LIN {X 0,Y 210.674,Z 740.227,A -85,B 0,C 180,E1 4144.705,E2 4144.705} C_VEL
LIN {X 0,Y 221.818,Z 721.614,A -85,B 0,C 180,E1 4143.81,E2 4143.81} C_VEL
LIN {X 0,Y 225.35,Z 714.922,A -85,B 0,C 180,E1 4143.336,E2 4143.336} C_VEL
LIN {X 0,Y 232.907,Z 698.102,A -85,B 0,C 180,E1 4141.321,E2 4141.321} C_VEL
LIN {X 0,Y 235.66,Z 691.099,A -85,B 0,C 180,E1 4140.884,E2 4140.884} C_VEL
LIN {X 0,Y 242.843,Z 670.512,A -85,B 0,C 180,E1 4140.52,E2 4140.52} C_VEL
LIN {X 0,Y 247.959,Z 650.095,A -85,B 0,C 180,E1 4140.233,E2 4140.233} C_VEL
LIN {X 0,Y 251.406,Z 630.033,A -85,B 0,C 180,E1 4139.968,E2 4139.968} C_VEL
LIN {X 0,Y 253.666,Z 611.872,A -85,B 0,C 180,E1 4139.728,E2 4139.728} C_VEL
LIN {X 0,Y 254.145,Z 615.413,A -85,B 0,C 180,E1 4134.932,E2 4134.932} C_VEL
LIN {X 0,Y 255.029,Z 619.345,A -85,B 0,C 180,E1 4132.123,E2 4132.123} C_VEL
LIN {X 0,Y 260.484,Z 634.906,A -85,B 0,C 180,E1 4123.968,E2 4123.968} C_VEL
LIN {X 0,Y 268.032,Z 645.56,A -85,B 0,C 180,E1 4117.878,E2 4117.878} C_VEL
LIN {X 0,Y 279.58,Z 655.999,A -85,B 0,C 180,E1 4111.494,E2 4111.494} C_VEL
LIN {X 0,Y 288.035,Z 662.589,A -85,B 0,C 180,E1 4107.697,E2 4107.697} C_VEL
LIN {X 0,Y 293.255,Z 666.559,A -85,B 0,C 180,E1 4105.252,E2 4105.252} C_VEL
LIN {X 0,Y 299.992,Z 671.93,A -85,B 0,C 180,E1 4101.864,E2 4101.864} C_VEL
LIN {X 0,Y 304.317,Z 675.457,A -85,B 0,C 180,E1 4099.555,E2 4099.555} C_VEL
LIN {X 0,Y 310.73,Z 680.537,A -85,B 0,C 180,E1 4095.985,E2 4095.985} C_VEL
LIN {X 0,Y 314.599,Z 683.638,A -85,B 0,C 180,E1 4093.71,E2 4093.71} C_VEL
LIN {X 0,Y 320.356,Z 688.374,A -85,B 0,C 180,E1 4090.14,E2 4090.14} C_VEL
LIN {X 0,Y 324.684,Z 691.53,A -85,B 0,C 180,E1 4087.347,E2 4087.347} C_VEL
LIN {X 0,Y 329.45,Z 695.655,A -85,B 0,C 180,E1 4083.946,E2 4083.946} C_VEL
LIN {X 0,Y 334.291,Z 698.905,A -85,B 0,C 180,E1 4080.362,E2 4080.362} C_VEL
LIN {X 0,Y 336.58,Z 700.785,A -85,B 0,C 180,E1 4078.464,E2 4078.464} C_VEL
LIN {X 0,Y 340.334,Z 704.161,A -85,B 0,C 180,E1 4075.027,E2 4075.027} C_VEL
LIN {X 0,Y 343.918,Z 706.626,A -85,B 0,C 180,E1 4071.488,E2 4071.488} C_VEL
LIN {X 0,Y 347.168,Z 708.204,A -85,B 0,C 180,E1 4067.948,E2 4067.948} C_VEL
LIN {X 0,Y 348.332,Z 709.173,A -85,B 0,C 180,E1 4066.337,E2 4066.337} C_VEL
LIN {X 0,Y 350.261,Z 711.431,A -85,B 0,C 180,E1 4063.033,E2 4063.033} C_VEL
LIN {X 0,Y 351.887,Z 712.957,A -85,B 0,C 180,E1 4059.651,E2 4059.651} C_VEL
LIN {X 0,Y 353.094,Z 713.879,A -85,B 0,C 180,E1 4056.34,E2 4056.34} C_VEL
LIN {X 0,Y 353.771,Z 714.356,A -85,B 0,C 180,E1 4053.078,E2 4053.078} C_VEL
LIN {X 0,Y 353.955,Z 714.518,A -85,B 0,C 180,E1 4049.676,E2 4049.676} C_VEL
LIN {X 0,Y 353.709,Z 714.308,A -85,B 0,C 180,E1 4046.435,E2 4046.435} C_VEL
LIN {X 0,Y 352.933,Z 713.762,A -85,B 0,C 180,E1 4043.167,E2 4043.167} C_VEL
LIN {X 0,Y 351.648,Z 712.791,A -85,B 0,C 180,E1 4039.847,E2 4039.847} C_VEL
LIN {X 0,Y 349.965,Z 711.152,A -85,B 0,C 180,E1 4036.451,E2 4036.451} C_VEL
LIN {X 0,Y 347.988,Z 708.725,A -85,B 0,C 180,E1 4033.131,E2 4033.131} C_VEL
LIN {X 0,Y 345.166,Z 707.3,A -85,B 0,C 180,E1 4029.836,E2 4029.836} C_VEL
LIN {X 0,Y 341.961,Z 705.369,A -85,B 0,C 180,E1 4026.569,E2 4026.569} C_VEL
LIN {X 0,Y 338.532,Z 702.666,A -85,B 0,C 180,E1 4023.326,E2 4023.326} C_VEL
LIN {X 0,Y 334.734,Z 699.159,A -85,B 0,C 180,E1 4020.002,E2 4020.002} C_VEL
LIN {X 0,Y 330.098,Z 696.163,A -85,B 0,C 180,E1 4016.547,E2 4016.547} C_VEL
LIN {X 0,Y 325.217,Z 692.068,A -85,B 0,C 180,E1 4013.05,E2 4013.05} C_VEL
LIN {X 0,Y 322.331,Z 689.725,A -85,B 0,C 180,E1 4011.114,E2 4011.114} C_VEL
LIN {X 0,Y 316.916,Z 685.673,A -85,B 0,C 180,E1 4007.715,E2 4007.715} C_VEL
LIN {X 0,Y 311.447,Z 681.018,A -85,B 0,C 180,E1 4004.401,E2 4004.401} C_VEL
LIN {X 0,Y 305.202,Z 676.225,A -85,B 0,C 180,E1 4000.921,E2 4000.921} C_VEL
LIN {X 0,Y 300.242,Z 672.107,A -85,B 0,C 180,E1 3998.259,E2 3998.259} C_VEL
LIN {X 0,Y 293.548,Z 666.815,A -85,B 0,C 180,E1 3994.892,E2 3994.892} C_VEL
LIN {X 0,Y 288.653,Z 663.022,A -85,B 0,C 180,E1 3992.578,E2 3992.578} C_VEL
LIN {X 0,Y 280.59,Z 656.799,A -85,B 0,C 180,E1 3988.975,E2 3988.975} C_VEL
LIN {X 0,Y 270.966,Z 648.453,A -85,B 0,C 180,E1 3983.936,E2 3983.936} C_VEL
LIN {X 0,Y 263.336,Z 639.521,A -85,B 0,C 180,E1 3978.587,E2 3978.587} C_VEL
LIN {X 0,Y 257.411,Z 627.943,A -85,B 0,C 180,E1 3972.325,E2 3972.325} C_VEL
LIN {X 0,Y 254.738,Z 618.098,A -85,B 0,C 180,E1 3967.092,E2 3967.092} C_VEL
LIN {X 0,Y 253.972,Z 614.598,A -85,B 0,C 180,E1 3964.28,E2 3964.28} C_VEL
LIN {X 0,Y 253.666,Z 611.872,A -85,B 0,C 180,E1 3960.272,E2 3960.272} C_VEL
LIN {X 0,Y 249.3,Z 643.642,A -85,B 0,C 180,E1 3959.853,E2 3959.853} C_VEL
LIN {X 0,Y 244.621,Z 664.019,A -85,B 0,C 180,E1 3959.573,E2 3959.573} C_VEL
LIN {X 0,Y 238.978,Z 682.281,A -85,B 0,C 180,E1 3959.285,E2 3959.285} C_VEL
LIN {X 0,Y 230.509,Z 703.314,A -85,B 0,C 180,E1 3958.824,E2 3958.824} C_VEL
LIN {X 0,Y 222.058,Z 720.216,A -85,B 0,C 180,E1 3958.313,E2 3958.313} C_VEL
LIN {X 0,Y 211.154,Z 738.544,A -85,B 0,C 180,E1 3957.565,E2 3957.565} C_VEL
LIN {X 0,Y 199.308,Z 755.025,A -85,B 0,C 180,E1 3956.64,E2 3956.64} C_VEL
LIN {X 0,Y 188.015,Z 768.679,A -85,B 0,C 180,E1 3955.629,E2 3955.629} C_VEL
LIN {X 0,Y 173.879,Z 783.577,A -85,B 0,C 180,E1 3954.14,E2 3954.14} C_VEL
LIN {X 0,Y 159.406,Z 796.517,A -85,B 0,C 180,E1 3952.311,E2 3952.311} C_VEL
LIN {X 0,Y 146.082,Z 807.005,A -85,B 0,C 180,E1 3950.256,E2 3950.256} C_VEL
LIN {X 0,Y 129.637,Z 818.368,A -85,B 0,C 180,E1 3947.057,E2 3947.057} C_VEL
LIN {X 0,Y 113.071,Z 827.981,A -85,B 0,C 180,E1 3942.744,E2 3942.744} C_VEL
LIN {X 0,Y 99.321,Z 834.97,A -85,B 0,C 180,E1 3937.839,E2 3937.839} C_VEL
LIN {X 0,Y 83.5,Z 842.05,A -85,B 0,C 180,E1 3929.556,E2 3929.556} C_VEL
LIN {X 0,Y 69.946,Z 847.19,A -85,B 0,C 180,E1 3917.745,E2 3917.745} C_VEL
LIN {X 0,Y 61.606,Z 850.22,A -85,B 0,C 180,E1 3904.613,E2 3904.613} C_VEL
LIN {X 0,Y 56.485,Z 852.404,A -85,B 0,C 180,E1 3885.397,E2 3885.397} C_VEL
LIN {X 0,Y 56.061,Z 852.878,A -85,B 0,C 180,E1 3871.022,E2 3871.022} C_VEL
LIN {X 0,Y 56.17,Z 852.551,A -85,B 0,C 180,E1 3858.448,E2 3858.448} C_VEL
LIN {X 0,Y 60.475,Z 850.675,A -85,B 0,C 180,E1 3838.058,E2 3838.058} C_VEL
LIN {X 0,Y 68.915,Z 847.568,A -85,B 0,C 180,E1 3823.497,E2 3823.497} C_VEL
LIN {X 0,Y 79.87,Z 843.421,A -85,B 0,C 180,E1 3812.995,E2 3812.995} C_VEL
LIN {X 0,Y 95.202,Z 836.983,A -85,B 0,C 180,E1 3803.979,E2 3803.979} C_VEL
LIN {X 0,Y 111.312,Z 828.923,A -85,B 0,C 180,E1 3797.803,E2 3797.803} C_VEL
LIN {X 0,Y 125.885,Z 820.608,A -85,B 0,C 180,E1 3793.804,E2 3793.804} C_VEL
LIN {X 0,Y 143.255,Z 809.115,A -85,B 0,C 180,E1 3790.235,E2 3790.235} C_VEL
LIN {X 0,Y 157.491,Z 798.103,A -85,B 0,C 180,E1 3787.96,E2 3787.96} C_VEL
LIN {X 0,Y 170.969,Z 786.254,A -85,B 0,C 180,E1 3786.195,E2 3786.195} C_VEL
LIN {X 0,Y 186.547,Z 770.362,A -85,B 0,C 180,E1 3784.515,E2 3784.515} C_VEL
LIN {X 0,Y 198.324,Z 756.287,A -85,B 0,C 180,E1 3783.443,E2 3783.443} C_VEL
LIN {X 0,Y 209.671,Z 740.706,A -85,B 0,C 180,E1 3782.543,E2 3782.543} C_VEL
LIN {X 0,Y 221.065,Z 722.057,A -85,B 0,C 180,E1 3781.751,E2 3781.751} C_VEL
LIN {X 0,Y 229.514,Z 705.439,A -85,B 0,C 180,E1 3781.232,E2 3781.232} C_VEL
LIN {X 0,Y 235.66,Z 691.099,A -85,B 0,C 180,E1 3780.884,E2 3780.884} C_VEL
LIN {X 0,Y 238.036,Z 684.989,A -85,B 0,C 180,E1 3780.593,E2 3780.593} C_VEL
LIN {X 0,Y 244.118,Z 666.072,A -85,B 0,C 180,E1 3778.809,E2 3778.809} C_VEL
LIN {X 0,Y 246.08,Z 658.696,A -85,B 0,C 180,E1 3778.485,E2 3778.485} C_VEL
LIN {X 0,Y 250.367,Z 637.413,A -85,B 0,C 180,E1 3778.231,E2 3778.231} C_VEL
LIN {X 0,Y 252.664,Z 621.011,A -85,B 0,C 180,E1 3778.026,E2 3778.026} C_VEL
LIN {X 0,Y 253.065,Z 623.238,A -85,B 0,C 180,E1 3775.251,E2 3775.251} C_VEL
LIN {X 0,Y 253.864,Z 627.304,A -85,B 0,C 180,E1 3772.429,E2 3772.429} C_VEL
LIN {X 0,Y 258.424,Z 642.042,A -85,B 0,C 180,E1 3764.642,E2 3764.642} C_VEL
LIN {X 0,Y 265.618,Z 652.99,A -85,B 0,C 180,E1 3758.248,E2 3758.248} C_VEL
LIN {X 0,Y 276.691,Z 663.352,A -85,B 0,C 180,E1 3751.758,E2 3751.758} C_VEL
LIN {X 0,Y 286.024,Z 670.633,A -85,B 0,C 180,E1 3747.442,E2 3747.442} C_VEL
LIN {X 0,Y 291.129,Z 674.665,A -85,B 0,C 180,E1 3745.015,E2 3745.015} C_VEL
LIN {X 0,Y 297.886,Z 679.891,A -85,B 0,C 180,E1 3741.628,E2 3741.628} C_VEL
LIN {X 0,Y 304.458,Z 685.399,A -85,B 0,C 180,E1 3738.078,E2 3738.078} C_VEL
LIN {X 0,Y 310.736,Z 690.084,A -85,B 0,C 180,E1 3734.543,E2 3734.543} C_VEL
LIN {X 0,Y 316.536,Z 695.023,A -85,B 0,C 180,E1 3730.997,E2 3730.997} C_VEL
LIN {X 0,Y 321.866,Z 698.858,A -85,B 0,C 180,E1 3727.632,E2 3727.632} C_VEL
LIN {X 0,Y 326.947,Z 703.244,A -85,B 0,C 180,E1 3724.03,E2 3724.03} C_VEL
LIN {X 0,Y 331.613,Z 706.372,A -85,B 0,C 180,E1 3720.633,E2 3720.633} C_VEL
LIN {X 0,Y 333.853,Z 708.095,A -85,B 0,C 180,E1 3718.827,E2 3718.827} C_VEL
LIN {X 0,Y 337.827,Z 711.687,A -85,B 0,C 180,E1 3715.225,E2 3715.225} C_VEL
LIN {X 0,Y 341.357,Z 714.12,A -85,B 0,C 180,E1 3711.826,E2 3711.826} C_VEL
LIN {X 0,Y 344.675,Z 715.784,A -85,B 0,C 180,E1 3708.257,E2 3708.257} C_VEL
LIN {X 0,Y 345.95,Z 716.669,A -85,B 0,C 180,E1 3706.626,E2 3706.626} C_VEL
LIN {X 0,Y 347.815,Z 718.903,A -85,B 0,C 180,E1 3703.464,E2 3703.464} C_VEL
LIN {X 0,Y 349.513,Z 720.522,A -85,B 0,C 180,E1 3700.049,E2 3700.049} C_VEL
LIN {X 0,Y 350.807,Z 721.495,A -85,B 0,C 180,E1 3696.711,E2 3696.711} C_VEL
LIN {X 0,Y 351.51,Z 722.006,A -85,B 0,C 180,E1 3693.424,E2 3693.424} C_VEL
LIN {X 0,Y 351.766,Z 722.221,A -85,B 0,C 180,E1 3690,E2 3690} C_VEL
LIN {X 0,Y 351.591,Z 722.033,A -85,B 0,C 180,E1 3686.74,E2 3686.74} C_VEL
LIN {X 0,Y 350.787,Z 721.516,A -85,B 0,C 180,E1 3683.453,E2 3683.453} C_VEL
LIN {X 0,Y 349.505,Z 720.527,A -85,B 0,C 180,E1 3679.95,E2 3679.95} C_VEL
LIN {X 0,Y 347.971,Z 719.018,A -85,B 0,C 180,E1 3676.711,E2 3676.711} C_VEL
LIN {X 0,Y 345.922,Z 716.659,A -85,B 0,C 180,E1 3673.373,E2 3673.373} C_VEL
LIN {X 0,Y 344.622,Z 715.769,A -85,B 0,C 180,E1 3671.74,E2 3671.74} C_VEL
LIN {X 0,Y 341.289,Z 714.097,A -85,B 0,C 180,E1 3668.158,E2 3668.158} C_VEL
LIN {X 0,Y 337.789,Z 711.674,A -85,B 0,C 180,E1 3664.772,E2 3664.772} C_VEL
LIN {X 0,Y 334.098,Z 708.347,A -85,B 0,C 180,E1 3661.392,E2 3661.392} C_VEL
LIN {X 0,Y 331.89,Z 706.536,A -85,B 0,C 180,E1 3659.595,E2 3659.595} C_VEL
LIN {X 0,Y 327.39,Z 703.585,A -85,B 0,C 180,E1 3656.292,E2 3656.292} C_VEL
LIN {X 0,Y 322.48,Z 699.458,A -85,B 0,C 180,E1 3652.801,E2 3652.801} C_VEL
LIN {X 0,Y 319.198,Z 696.92,A -85,B 0,C 180,E1 3650.67,E2 3650.67} C_VEL
LIN {X 0,Y 313.547,Z 692.596,A -85,B 0,C 180,E1 3647.159,E2 3647.159} C_VEL
LIN {X 0,Y 308.746,Z 688.532,A -85,B 0,C 180,E1 3644.301,E2 3644.301} C_VEL
LIN {X 0,Y 302.375,Z 683.685,A -85,B 0,C 180,E1 3640.781,E2 3640.781} C_VEL
LIN {X 0,Y 297.355,Z 679.512,A -85,B 0,C 180,E1 3638.085,E2 3638.085} C_VEL
LIN {X 0,Y 290.395,Z 674.023,A -85,B 0,C 180,E1 3634.605,E2 3634.605} C_VEL
LIN {X 0,Y 284.812,Z 669.781,A -85,B 0,C 180,E1 3631.999,E2 3631.999} C_VEL
LIN {X 0,Y 272.035,Z 659.617,A -85,B 0,C 180,E1 3625.808,E2 3625.808} C_VEL
LIN {X 0,Y 261.158,Z 646.993,A -85,B 0,C 180,E1 3618.17,E2 3618.17} C_VEL
LIN {X 0,Y 255.873,Z 635.734,A -85,B 0,C 180,E1 3611.942,E2 3611.942} C_VEL
LIN {X 0,Y 253.53,Z 625.643,A -85,B 0,C 180,E1 3606.557,E2 3606.557} C_VEL
LIN {X 0,Y 252.891,Z 622.329,A -85,B 0,C 180,E1 3603.844,E2 3603.844} C_VEL
LIN {X 0,Y 252.634,Z 621.243,A -85,B 0,C 180,E1 3601.964,E2 3601.964} C_VEL
LIN {X 0,Y 248.718,Z 646.779,A -85,B 0,C 180,E1 3601.657,E2 3601.657} C_VEL
LIN {X 0,Y 244.033,Z 666.201,A -85,B 0,C 180,E1 3601.423,E2 3601.423} C_VEL
LIN {X 0,Y 237.507,Z 686.316,A -85,B 0,C 180,E1 3601.144,E2 3601.144} C_VEL
LIN {X 0,Y 229.482,Z 705.211,A -85,B 0,C 180,E1 3600.777,E2 3600.777} C_VEL
LIN {X 0,Y 220.465,Z 722.748,A -85,B 0,C 180,E1 3600.311,E2 3600.311} C_VEL
LIN {X 0,Y 208.618,Z 741.685,A -85,B 0,C 180,E1 3599.614,E2 3599.614} C_VEL
LIN {X 0,Y 197.505,Z 756.683,A -85,B 0,C 180,E1 3598.863,E2 3598.863} C_VEL
LIN {X 0,Y 184.072,Z 772.379,A -85,B 0,C 180,E1 3597.808,E2 3597.808} C_VEL
LIN {X 0,Y 169.299,Z 786.908,A -85,B 0,C 180,E1 3596.431,E2 3596.431} C_VEL
LIN {X 0,Y 155.594,Z 798.659,A -85,B 0,C 180,E1 3594.88,E2 3594.88} C_VEL
LIN {X 0,Y 138.984,Z 811.022,A -85,B 0,C 180,E1 3592.542,E2 3592.542} C_VEL
LIN {X 0,Y 122.989,Z 821.059,A -85,B 0,C 180,E1 3589.628,E2 3589.628} C_VEL
LIN {X 0,Y 108.169,Z 829.154,A -85,B 0,C 180,E1 3586.057,E2 3586.057} C_VEL
LIN {X 0,Y 90.447,Z 837.455,A -85,B 0,C 180,E1 3579.987,E2 3579.987} C_VEL
LIN {X 0,Y 74.938,Z 843.452,A -85,B 0,C 180,E1 3571.712,E2 3571.712} C_VEL
LIN {X 0,Y 62.908,Z 847.538,A -85,B 0,C 180,E1 3561.149,E2 3561.149} C_VEL
LIN {X 0,Y 52.118,Z 850.964,A -85,B 0,C 180,E1 3542.49,E2 3542.49} C_VEL
LIN {X 0,Y 48.181,Z 852.354,A -85,B 0,C 180,E1 3521.977,E2 3521.977} C_VEL
LIN {X 0,Y 48.051,Z 852.632,A -85,B 0,C 180,E1 3508.42,E2 3508.42} C_VEL
LIN {X 0,Y 49.054,Z 851.983,A -85,B 0,C 180,E1 3489.727,E2 3489.727} C_VEL
LIN {X 0,Y 55.075,Z 849.978,A -85,B 0,C 180,E1 3470.551,E2 3470.551} C_VEL
LIN {X 0,Y 64.861,Z 846.901,A -85,B 0,C 180,E1 3456.719,E2 3456.719} C_VEL
LIN {X 0,Y 79.842,Z 841.738,A -85,B 0,C 180,E1 3445.233,E2 3445.233} C_VEL
LIN {X 0,Y 96.521,Z 834.727,A -85,B 0,C 180,E1 3437.637,E2 3437.637} C_VEL
LIN {X 0,Y 110.912,Z 827.74,A -85,B 0,C 180,E1 3433.201,E2 3433.201} C_VEL
LIN {X 0,Y 127.705,Z 818.334,A -85,B 0,C 180,E1 3429.432,E2 3429.432} C_VEL
LIN {X 0,Y 144.922,Z 806.767,A -85,B 0,C 180,E1 3426.554,E2 3426.554} C_VEL
LIN {X 0,Y 159.497,Z 795.486,A -85,B 0,C 180,E1 3424.646,E2 3424.646} C_VEL
LIN {X 0,Y 176.194,Z 780.394,A -85,B 0,C 180,E1 3422.893,E2 3422.893} C_VEL
LIN {X 0,Y 189.058,Z 766.76,A -85,B 0,C 180,E1 3421.775,E2 3421.775} C_VEL
LIN {X 0,Y 201.986,Z 751.007,A -85,B 0,C 180,E1 3420.824,E2 3420.824} C_VEL
LIN {X 0,Y 213.963,Z 733.546,A -85,B 0,C 180,E1 3420.055,E2 3420.055} C_VEL
LIN {X 0,Y 222.968,Z 718.144,A -85,B 0,C 180,E1 3419.551,E2 3419.551} C_VEL
LIN {X 0,Y 231.988,Z 699.85,A -85,B 0,C 180,E1 3419.105,E2 3419.105} C_VEL
LIN {X 0,Y 239.765,Z 679.826,A -85,B 0,C 180,E1 3418.756,E2 3418.756} C_VEL
LIN {X 0,Y 245.667,Z 660.249,A -85,B 0,C 180,E1 3418.504,E2 3418.504} C_VEL
LIN {X 0,Y 246.08,Z 658.696,A -85,B 0,C 180,E1 3418.485,E2 3418.485} C_VEL
LIN {X 0,Y 247.29,Z 653.76,A -85,B 0,C 180,E1 3418.194,E2 3418.194} C_VEL
LIN {X 0,Y 250.073,Z 641.294,A -85,B 0,C 180,E1 3416.626,E2 3416.626} C_VEL
LIN {X 0,Y 250.775,Z 636.973,A -85,B 0,C 180,E1 3416.396,E2 3416.396} C_VEL
LIN {X 0,Y 251.823,Z 630.238,A -85,B 0,C 180,E1 3416.317,E2 3416.317} C_VEL
LIN {X 0,Y 252.307,Z 633.846,A -85,B 0,C 180,E1 3413.525,E2 3413.525} C_VEL
LIN {X 0,Y 256.15,Z 649.128,A -85,B 0,C 180,E1 3405.313,E2 3405.313} C_VEL
LIN {X 0,Y 263,Z 660.366,A -85,B 0,C 180,E1 3398.606,E2 3398.606} C_VEL
LIN {X 0,Y 282.175,Z 677.465,A -85,B 0,C 180,E1 3387.906,E2 3387.906} C_VEL
LIN {X 0,Y 287.738,Z 681.797,A -85,B 0,C 180,E1 3385.271,E2 3385.271} C_VEL
LIN {X 0,Y 294.58,Z 687.092,A -85,B 0,C 180,E1 3381.863,E2 3381.863} C_VEL
LIN {X 0,Y 301.39,Z 692.769,A -85,B 0,C 180,E1 3378.193,E2 3378.193} C_VEL
LIN {X 0,Y 308.027,Z 697.735,A -85,B 0,C 180,E1 3374.517,E2 3374.517} C_VEL
LIN {X 0,Y 314.137,Z 702.845,A -85,B 0,C 180,E1 3370.771,E2 3370.771} C_VEL
LIN {X 0,Y 319.077,Z 706.411,A -85,B 0,C 180,E1 3367.664,E2 3367.664} C_VEL
LIN {X 0,Y 323.715,Z 710.397,A -85,B 0,C 180,E1 3364.417,E2 3364.417} C_VEL
LIN {X 0,Y 328.566,Z 713.706,A -85,B 0,C 180,E1 3360.912,E2 3360.912} C_VEL
LIN {X 0,Y 330.854,Z 715.363,A -85,B 0,C 180,E1 3359.113,E2 3359.113} C_VEL
LIN {X 0,Y 334.802,Z 718.941,A -85,B 0,C 180,E1 3355.617,E2 3355.617} C_VEL
LIN {X 0,Y 338.558,Z 721.576,A -85,B 0,C 180,E1 3352.007,E2 3352.007} C_VEL
LIN {X 0,Y 341.818,Z 723.237,A -85,B 0,C 180,E1 3348.592,E2 3348.592} C_VEL
LIN {X 0,Y 343.348,Z 724.234,A -85,B 0,C 180,E1 3346.689,E2 3346.689} C_VEL
LIN {X 0,Y 345.306,Z 726.538,A -85,B 0,C 180,E1 3343.394,E2 3343.394} C_VEL
LIN {X 0,Y 346.929,Z 728.083,A -85,B 0,C 180,E1 3340.125,E2 3340.125} C_VEL
LIN {X 0,Y 348.245,Z 729.07,A -85,B 0,C 180,E1 3336.76,E2 3336.76} C_VEL
LIN {X 0,Y 348.97,Z 729.591,A -85,B 0,C 180,E1 3333.449,E2 3333.449} C_VEL
LIN {X 0,Y 349.227,Z 729.808,A -85,B 0,C 180,E1 3330,E2 3330} C_VEL
LIN {X 0,Y 349.044,Z 729.616,A -85,B 0,C 180,E1 3326.716,E2 3326.716} C_VEL
LIN {X 0,Y 348.22,Z 729.081,A -85,B 0,C 180,E1 3323.357,E2 3323.357} C_VEL
LIN {X 0,Y 347.033,Z 728.155,A -85,B 0,C 180,E1 3320.046,E2 3320.046} C_VEL
LIN {X 0,Y 345.409,Z 726.629,A -85,B 0,C 180,E1 3316.781,E2 3316.781} C_VEL
LIN {X 0,Y 343.365,Z 724.308,A -85,B 0,C 180,E1 3313.42,E2 3313.42} C_VEL
LIN {X 0,Y 342.086,Z 723.358,A -85,B 0,C 180,E1 3311.754,E2 3311.754} C_VEL
LIN {X 0,Y 339.141,Z 721.922,A -85,B 0,C 180,E1 3308.558,E2 3308.558} C_VEL
LIN {X 0,Y 335.405,Z 719.421,A -85,B 0,C 180,E1 3304.957,E2 3304.957} C_VEL
LIN {X 0,Y 331.598,Z 716.116,A -85,B 0,C 180,E1 3301.55,E2 3301.55} C_VEL
LIN {X 0,Y 329.152,Z 714.04,A -85,B 0,C 180,E1 3299.517,E2 3299.517} C_VEL
LIN {X 0,Y 324.617,Z 711.095,A -85,B 0,C 180,E1 3296.247,E2 3296.247} C_VEL
LIN {X 0,Y 319.801,Z 707.113,A -85,B 0,C 180,E1 3292.851,E2 3292.851} C_VEL
LIN {X 0,Y 316.533,Z 704.497,A -85,B 0,C 180,E1 3290.688,E2 3290.688} C_VEL
LIN {X 0,Y 310.786,Z 700.181,A -85,B 0,C 180,E1 3287.166,E2 3287.166} C_VEL
LIN {X 0,Y 305.337,Z 695.643,A -85,B 0,C 180,E1 3283.949,E2 3283.949} C_VEL
LIN {X 0,Y 298.936,Z 690.73,A -85,B 0,C 180,E1 3280.442,E2 3280.442} C_VEL
LIN {X 0,Y 294.204,Z 686.831,A -85,B 0,C 180,E1 3277.948,E2 3277.948} C_VEL
LIN {X 0,Y 287.367,Z 681.475,A -85,B 0,C 180,E1 3274.537,E2 3274.537} C_VEL
LIN {X 0,Y 282.161,Z 677.461,A -85,B 0,C 180,E1 3272.096,E2 3272.096} C_VEL
LIN {X 0,Y 269.586,Z 667.398,A -85,B 0,C 180,E1 3265.823,E2 3265.823} C_VEL
LIN {X 0,Y 258.829,Z 654.428,A -85,B 0,C 180,E1 3257.757,E2 3257.757} C_VEL
LIN {X 0,Y 253.962,Z 642.615,A -85,B 0,C 180,E1 3251.112,E2 3251.112} C_VEL
LIN {X 0,Y 252.196,Z 633.003,A -85,B 0,C 180,E1 3245.906,E2 3245.906} C_VEL
LIN {X 0,Y 251.811,Z 630.349,A -85,B 0,C 180,E1 3243.676,E2 3243.676} C_VEL
LIN {X 0,Y 248.294,Z 650.213,A -85,B 0,C 180,E1 3243.465,E2 3243.465} C_VEL
LIN {X 0,Y 242.944,Z 670.96,A -85,B 0,C 180,E1 3243.255,E2 3243.255} C_VEL
LIN {X 0,Y 235.786,Z 691.065,A -85,B 0,C 180,E1 3243.015,E2 3243.015} C_VEL
LIN {X 0,Y 228.219,Z 708.169,A -85,B 0,C 180,E1 3242.725,E2 3242.725} C_VEL
LIN {X 0,Y 217.495,Z 727.891,A -85,B 0,C 180,E1 3242.265,E2 3242.265} C_VEL
LIN {X 0,Y 207.061,Z 743.799,A -85,B 0,C 180,E1 3241.749,E2 3241.749} C_VEL
LIN {X 0,Y 195,Z 759.6,A -85,B 0,C 180,E1 3241.062,E2 3241.062} C_VEL
LIN {X 0,Y 180.469,Z 775.658,A -85,B 0,C 180,E1 3240.092,E2 3240.092} C_VEL
LIN {X 0,Y 166.996,Z 788.453,A -85,B 0,C 180,E1 3239.019,E2 3239.019} C_VEL
LIN {X 0,Y 151.122,Z 801.569,A -85,B 0,C 180,E1 3237.466,E2 3237.466} C_VEL
LIN {X 0,Y 134.41,Z 813.162,A -85,B 0,C 180,E1 3235.402,E2 3235.402} C_VEL
LIN {X 0,Y 118.889,Z 822.451,A -85,B 0,C 180,E1 3232.911,E2 3232.911} C_VEL
LIN {X 0,Y 100.851,Z 831.67,A -85,B 0,C 180,E1 3228.956,E2 3228.956} C_VEL
LIN {X 0,Y 83.492,Z 838.899,A -85,B 0,C 180,E1 3223.337,E2 3223.337} C_VEL
LIN {X 0,Y 68.829,Z 844.066,A -85,B 0,C 180,E1 3215.962,E2 3215.962} C_VEL
LIN {X 0,Y 52.656,Z 848.823,A -85,B 0,C 180,E1 3201.123,E2 3201.123} C_VEL
LIN {X 0,Y 43.384,Z 851.188,A -85,B 0,C 180,E1 3182.009,E2 3182.009} C_VEL
LIN {X 0,Y 40.091,Z 852.214,A -85,B 0,C 180,E1 3160.054,E2 3160.054} C_VEL
LIN {X 0,Y 40.029,Z 852.374,A -85,B 0,C 180,E1 3147.137,E2 3147.137} C_VEL
LIN {X 0,Y 42.07,Z 851.558,A -85,B 0,C 180,E1 3123.157,E2 3123.157} C_VEL
LIN {X 0,Y 49.881,Z 849.513,A -85,B 0,C 180,E1 3103.027,E2 3103.027} C_VEL
LIN {X 0,Y 62.065,Z 846.165,A -85,B 0,C 180,E1 3088.944,E2 3088.944} C_VEL
LIN {X 0,Y 79.965,Z 840.246,A -85,B 0,C 180,E1 3078.148,E2 3078.148} C_VEL
LIN {X 0,Y 95.278,Z 834.085,A -85,B 0,C 180,E1 3072.598,E2 3072.598} C_VEL
LIN {X 0,Y 111.231,Z 826.559,A -85,B 0,C 180,E1 3068.598,E2 3068.598} C_VEL
LIN {X 0,Y 130.508,Z 815.646,A -85,B 0,C 180,E1 3065.166,E2 3065.166} C_VEL
LIN {X 0,Y 145.517,Z 805.602,A -85,B 0,C 180,E1 3063.168,E2 3063.168} C_VEL
LIN {X 0,Y 162.034,Z 792.845,A -85,B 0,C 180,E1 3061.43,E2 3061.43} C_VEL
LIN {X 0,Y 177.559,Z 778.57,A -85,B 0,C 180,E1 3060.123,E2 3060.123} C_VEL
LIN {X 0,Y 190.53,Z 764.791,A -85,B 0,C 180,E1 3059.214,E2 3059.214} C_VEL
LIN {X 0,Y 204.546,Z 747.356,A -85,B 0,C 180,E1 3058.387,E2 3058.387} C_VEL
LIN {X 0,Y 215.619,Z 730.893,A -85,B 0,C 180,E1 3057.82,E2 3057.82} C_VEL
LIN {X 0,Y 225.698,Z 713.295,A -85,B 0,C 180,E1 3057.378,E2 3057.378} C_VEL
LIN {X 0,Y 234.777,Z 693.553,A -85,B 0,C 180,E1 3057.021,E2 3057.021} C_VEL
LIN {X 0,Y 241.336,Z 675.883,A -85,B 0,C 180,E1 3056.796,E2 3056.796} C_VEL
LIN {X 0,Y 247.442,Z 654.174,A -85,B 0,C 180,E1 3056.576,E2 3056.576} C_VEL
LIN {X 0,Y 250.775,Z 636.973,A -85,B 0,C 180,E1 3056.396,E2 3056.396} C_VEL
LIN {X 0,Y 251.008,Z 635.871,A -85,B 0,C 180,E1 3056.158,E2 3056.158} C_VEL
LIN {X 0,Y 251.231,Z 635.803,A -85,B 0,C 180,E1 3055.473,E2 3055.473} C_VEL
LIN {X 0,Y 251.312,Z 637.609,A -85,B 0,C 180,E1 3054.477,E2 3054.477} C_VEL
LIN {X 0,Y 251.28,Z 645.589,A -85,B 0,C 180,E1 3051.782,E2 3051.782} C_VEL
LIN {X 0,Y 251.36,Z 646.438,A -85,B 0,C 180,E1 3051.363,E2 3051.363} C_VEL
LIN {X 0,Y 254.203,Z 657.281,A -85,B 0,C 180,E1 3045.315,E2 3045.315} C_VEL
LIN {X 0,Y 260.03,Z 667.519,A -85,B 0,C 180,E1 3039.059,E2 3039.059} C_VEL
LIN {X 0,Y 270.301,Z 677.852,A -85,B 0,C 180,E1 3032.232,E2 3032.232} C_VEL
LIN {X 0,Y 282.152,Z 687.144,A -85,B 0,C 180,E1 3026.453,E2 3026.453} C_VEL
LIN {X 0,Y 289.105,Z 692.824,A -85,B 0,C 180,E1 3023.017,E2 3023.017} C_VEL
LIN {X 0,Y 294.362,Z 696.919,A -85,B 0,C 180,E1 3020.329,E2 3020.329} C_VEL
LIN {X 0,Y 301.066,Z 702.252,A -85,B 0,C 180,E1 3016.66,E2 3016.66} C_VEL
LIN {X 0,Y 305.071,Z 705.329,A -85,B 0,C 180,E1 3014.415,E2 3014.415} C_VEL
LIN {X 0,Y 310.84,Z 710.095,A -85,B 0,C 180,E1 3010.912,E2 3010.912} C_VEL
LIN {X 0,Y 315.67,Z 713.531,A -85,B 0,C 180,E1 3007.913,E2 3007.913} C_VEL
LIN {X 0,Y 320.47,Z 717.665,A -85,B 0,C 180,E1 3004.566,E2 3004.566} C_VEL
LIN {X 0,Y 325.452,Z 721.055,A -85,B 0,C 180,E1 3001.024,E2 3001.024} C_VEL
LIN {X 0,Y 327.786,Z 722.736,A -85,B 0,C 180,E1 2999.212,E2 2999.212} C_VEL
LIN {X 0,Y 331.716,Z 726.305,A -85,B 0,C 180,E1 2995.704,E2 2995.704} C_VEL
LIN {X 0,Y 335.545,Z 728.983,A -85,B 0,C 180,E1 2992.052,E2 2992.052} C_VEL
LIN {X 0,Y 338.929,Z 730.698,A -85,B 0,C 180,E1 2988.578,E2 2988.578} C_VEL
LIN {X 0,Y 340.381,Z 731.645,A -85,B 0,C 180,E1 2986.781,E2 2986.781} C_VEL
LIN {X 0,Y 342.471,Z 734.047,A -85,B 0,C 180,E1 2983.335,E2 2983.335} C_VEL
LIN {X 0,Y 344.087,Z 735.588,A -85,B 0,C 180,E1 2979.977,E2 2979.977} C_VEL
LIN {X 0,Y 345.408,Z 736.585,A -85,B 0,C 180,E1 2976.482,E2 2976.482} C_VEL
LIN {X 0,Y 346.13,Z 737.076,A -85,B 0,C 180,E1 2973.312,E2 2973.312} C_VEL
LIN {X 0,Y 346.351,Z 737.273,A -85,B 0,C 180,E1 2970,E2 2970} C_VEL
LIN {X 0,Y 346.165,Z 737.091,A -85,B 0,C 180,E1 2966.854,E2 2966.854} C_VEL
LIN {X 0,Y 345.392,Z 736.588,A -85,B 0,C 180,E1 2963.518,E2 2963.518} C_VEL
LIN {X 0,Y 344.271,Z 735.7,A -85,B 0,C 180,E1 2960.303,E2 2960.303} C_VEL
LIN {X 0,Y 342.6,Z 734.203,A -85,B 0,C 180,E1 2957.014,E2 2957.014} C_VEL
LIN {X 0,Y 340.639,Z 731.993,A -85,B 0,C 180,E1 2953.634,E2 2953.634} C_VEL
LIN {X 0,Y 339.482,Z 730.93,A -85,B 0,C 180,E1 2951.986,E2 2951.986} C_VEL
LIN {X 0,Y 336.314,Z 729.439,A -85,B 0,C 180,E1 2948.734,E2 2948.734} C_VEL
LIN {X 0,Y 332.552,Z 726.969,A -85,B 0,C 180,E1 2945.108,E2 2945.108} C_VEL
LIN {X 0,Y 328.912,Z 723.869,A -85,B 0,C 180,E1 2941.809,E2 2941.809} C_VEL
LIN {X 0,Y 326.09,Z 721.427,A -85,B 0,C 180,E1 2939.475,E2 2939.475} C_VEL
LIN {X 0,Y 321.434,Z 718.407,A -85,B 0,C 180,E1 2936.134,E2 2936.134} C_VEL
LIN {X 0,Y 316.466,Z 714.306,A -85,B 0,C 180,E1 2932.656,E2 2932.656} C_VEL
LIN {X 0,Y 313.291,Z 711.785,A -85,B 0,C 180,E1 2930.574,E2 2930.574} C_VEL
LIN {X 0,Y 307.417,Z 707.395,A -85,B 0,C 180,E1 2927.021,E2 2927.021} C_VEL
LIN {X 0,Y 302.285,Z 703.076,A -85,B 0,C 180,E1 2923.981,E2 2923.981} C_VEL
LIN {X 0,Y 295.781,Z 698.16,A -85,B 0,C 180,E1 2920.454,E2 2920.454} C_VEL
LIN {X 0,Y 290.499,Z 693.827,A -85,B 0,C 180,E1 2917.664,E2 2917.664} C_VEL
LIN {X 0,Y 283.328,Z 688.17,A -85,B 0,C 180,E1 2914.119,E2 2914.119} C_VEL
LIN {X 0,Y 278.041,Z 684.177,A -85,B 0,C 180,E1 2911.657,E2 2911.657} C_VEL
LIN {X 0,Y 262.385,Z 670.162,A -85,B 0,C 180,E1 2902.742,E2 2902.742} C_VEL
LIN {X 0,Y 256.199,Z 661.62,A -85,B 0,C 180,E1 2897.242,E2 2897.242} C_VEL
LIN {X 0,Y 251.997,Z 650.11,A -85,B 0,C 180,E1 2890.621,E2 2890.621} C_VEL
LIN {X 0,Y 250.829,Z 640.57,A -85,B 0,C 180,E1 2885.401,E2 2885.401} C_VEL
LIN {X 0,Y 245.941,Z 662.213,A -85,B 0,C 180,E1 2885.207,E2 2885.207} C_VEL
LIN {X 0,Y 239.89,Z 681.604,A -85,B 0,C 180,E1 2885.049,E2 2885.049} C_VEL
LIN {X 0,Y 231.276,Z 702.629,A -85,B 0,C 180,E1 2884.814,E2 2884.814} C_VEL
LIN {X 0,Y 222.299,Z 720.186,A -85,B 0,C 180,E1 2884.535,E2 2884.535} C_VEL
LIN {X 0,Y 210.503,Z 739.297,A -85,B 0,C 180,E1 2884.103,E2 2884.103} C_VEL
LIN {X 0,Y 198.354,Z 755.584,A -85,B 0,C 180,E1 2883.585,E2 2883.585} C_VEL
LIN {X 0,Y 184.704,Z 771.333,A -85,B 0,C 180,E1 2882.897,E2 2882.897} C_VEL
LIN {X 0,Y 169.069,Z 786.433,A -85,B 0,C 180,E1 2881.949,E2 2881.949} C_VEL
LIN {X 0,Y 154.993,Z 798.185,A -85,B 0,C 180,E1 2880.905,E2 2880.905} C_VEL
LIN {X 0,Y 136.989,Z 811.06,A -85,B 0,C 180,E1 2879.218,E2 2879.218} C_VEL
LIN {X 0,Y 119.872,Z 821.265,A -85,B 0,C 180,E1 2877.111,E2 2877.111} C_VEL
LIN {X 0,Y 102.509,Z 830.09,A -85,B 0,C 180,E1 2874.193,E2 2874.193} C_VEL
LIN {X 0,Y 83.39,Z 837.984,A -85,B 0,C 180,E1 2869.472,E2 2869.472} C_VEL
LIN {X 0,Y 67.799,Z 843.242,A -85,B 0,C 180,E1 2863.447,E2 2863.447} C_VEL
LIN {X 0,Y 51.757,Z 847.692,A -85,B 0,C 180,E1 2852.7,E2 2852.7} C_VEL
LIN {X 0,Y 37.717,Z 850.761,A -85,B 0,C 180,E1 2831.507,E2 2831.507} C_VEL
LIN {X 0,Y 32.267,Z 851.943,A -85,B 0,C 180,E1 2804.353,E2 2804.353} C_VEL
LIN {X 0,Y 32.046,Z 852.168,A -85,B 0,C 180,E1 2788.212,E2 2788.212} C_VEL
LIN {X 0,Y 34.631,Z 851.411,A -85,B 0,C 180,E1 2758.689,E2 2758.689} C_VEL
LIN {X 0,Y 44.375,Z 849.344,A -85,B 0,C 180,E1 2735.793,E2 2735.793} C_VEL
LIN {X 0,Y 58.264,Z 845.994,A -85,B 0,C 180,E1 2722.08,E2 2722.08} C_VEL
LIN {X 0,Y 77.797,Z 840.006,A -85,B 0,C 180,E1 2712.385,E2 2712.385} C_VEL
LIN {X 0,Y 93.829,Z 833.846,A -85,B 0,C 180,E1 2707.694,E2 2707.694} C_VEL
LIN {X 0,Y 111.282,Z 825.849,A -85,B 0,C 180,E1 2704.214,E2 2704.214} C_VEL
LIN {X 0,Y 130.026,Z 815.407,A -85,B 0,C 180,E1 2701.568,E2 2701.568} C_VEL
LIN {X 0,Y 145.975,Z 804.886,A -85,B 0,C 180,E1 2699.882,E2 2699.882} C_VEL
LIN {X 0,Y 163.03,Z 791.771,A -85,B 0,C 180,E1 2698.473,E2 2698.473} C_VEL
LIN {X 0,Y 178.142,Z 777.924,A -85,B 0,C 180,E1 2697.475,E2 2697.475} C_VEL
LIN {X 0,Y 191.274,Z 764.045,A -85,B 0,C 180,E1 2696.755,E2 2696.755} C_VEL
LIN {X 0,Y 205.44,Z 746.412,A -85,B 0,C 180,E1 2696.103,E2 2696.103} C_VEL
LIN {X 0,Y 216.077,Z 730.659,A -85,B 0,C 180,E1 2695.681,E2 2695.681} C_VEL
LIN {X 0,Y 226.209,Z 713.053,A -85,B 0,C 180,E1 2695.339,E2 2695.339} C_VEL
LIN {X 0,Y 235.332,Z 693.321,A -85,B 0,C 180,E1 2695.066,E2 2695.066} C_VEL
LIN {X 0,Y 241.917,Z 675.658,A -85,B 0,C 180,E1 2694.897,E2 2694.897} C_VEL
LIN {X 0,Y 248.045,Z 653.984,A -85,B 0,C 180,E1 2694.726,E2 2694.726} C_VEL
LIN {X 0,Y 250.827,Z 640.601,A -85,B 0,C 180,E1 2694.578,E2 2694.578} C_VEL
LIN {X 0,Y 251.36,Z 646.438,A -85,B 0,C 180,E1 2691.363,E2 2691.363} C_VEL
LIN {X 0,Y 251.633,Z 650.208,A -85,B 0,C 180,E1 2689.822,E2 2689.822} C_VEL
LIN {X 0,Y 251.84,Z 663.238,A -85,B 0,C 180,E1 2686.023,E2 2686.023} C_VEL
LIN {X 0,Y 252.409,Z 666.32,A -85,B 0,C 180,E1 2684.694,E2 2684.694} C_VEL
LIN {X 0,Y 257.161,Z 674.934,A -85,B 0,C 180,E1 2679.291,E2 2679.291} C_VEL
LIN {X 0,Y 274.549,Z 691.382,A -85,B 0,C 180,E1 2668.384,E2 2668.384} C_VEL
LIN {X 0,Y 279.83,Z 695.427,A -85,B 0,C 180,E1 2665.89,E2 2665.89} C_VEL
LIN {X 0,Y 286.84,Z 700.928,A -85,B 0,C 180,E1 2662.424,E2 2662.424} C_VEL
LIN {X 0,Y 291.315,Z 704.57,A -85,B 0,C 180,E1 2660.087,E2 2660.087} C_VEL
LIN {X 0,Y 298.145,Z 709.837,A -85,B 0,C 180,E1 2656.415,E2 2656.415} C_VEL
LIN {X 0,Y 302.844,Z 713.661,A -85,B 0,C 180,E1 2653.71,E2 2653.71} C_VEL
LIN {X 0,Y 308.776,Z 718.29,A -85,B 0,C 180,E1 2650.118,E2 2650.118} C_VEL
LIN {X 0,Y 312.473,Z 721.005,A -85,B 0,C 180,E1 2647.8,E2 2647.8} C_VEL
LIN {X 0,Y 317.388,Z 725.148,A -85,B 0,C 180,E1 2644.394,E2 2644.394} C_VEL
LIN {X 0,Y 322.426,Z 728.504,A -85,B 0,C 180,E1 2640.819,E2 2640.819} C_VEL
LIN {X 0,Y 324.828,Z 730.417,A -85,B 0,C 180,E1 2638.898,E2 2638.898} C_VEL
LIN {X 0,Y 328.525,Z 733.693,A -85,B 0,C 180,E1 2635.605,E2 2635.605} C_VEL
LIN {X 0,Y 332.479,Z 736.403,A -85,B 0,C 180,E1 2631.894,E2 2631.894} C_VEL
LIN {X 0,Y 335.583,Z 737.964,A -85,B 0,C 180,E1 2628.689,E2 2628.689} C_VEL
LIN {X 0,Y 337.049,Z 738.884,A -85,B 0,C 180,E1 2626.9,E2 2626.9} C_VEL
LIN {X 0,Y 339.152,Z 741.31,A -85,B 0,C 180,E1 2623.424,E2 2623.424} C_VEL
LIN {X 0,Y 340.756,Z 742.842,A -85,B 0,C 180,E1 2620.14,E2 2620.14} C_VEL
LIN {X 0,Y 342.142,Z 743.882,A -85,B 0,C 180,E1 2616.544,E2 2616.544} C_VEL
LIN {X 0,Y 342.873,Z 744.38,A -85,B 0,C 180,E1 2613.511,E2 2613.511} C_VEL
LIN {X 0,Y 343.14,Z 744.6,A -85,B 0,C 180,E1 2610,E2 2610} C_VEL
LIN {X 0,Y 342.951,Z 744.432,A -85,B 0,C 180,E1 2606.992,E2 2606.992} C_VEL
LIN {X 0,Y 342.126,Z 743.883,A -85,B 0,C 180,E1 2603.437,E2 2603.437} C_VEL
LIN {X 0,Y 340.929,Z 742.952,A -85,B 0,C 180,E1 2600.132,E2 2600.132} C_VEL
LIN {X 0,Y 339.165,Z 741.353,A -85,B 0,C 180,E1 2596.707,E2 2596.707} C_VEL
LIN {X 0,Y 337.162,Z 739.033,A -85,B 0,C 180,E1 2593.268,E2 2593.268} C_VEL
LIN {X 0,Y 335.714,Z 738.026,A -85,B 0,C 180,E1 2591.418,E2 2591.418} C_VEL
LIN {X 0,Y 332.577,Z 736.47,A -85,B 0,C 180,E1 2588.245,E2 2588.245} C_VEL
LIN {X 0,Y 328.699,Z 733.842,A -85,B 0,C 180,E1 2584.587,E2 2584.587} C_VEL
LIN {X 0,Y 324.974,Z 730.573,A -85,B 0,C 180,E1 2581.243,E2 2581.243} C_VEL
LIN {X 0,Y 322.76,Z 728.697,A -85,B 0,C 180,E1 2579.429,E2 2579.429} C_VEL
LIN {X 0,Y 318.055,Z 725.651,A -85,B 0,C 180,E1 2576.071,E2 2576.071} C_VEL
LIN {X 0,Y 313.109,Z 721.612,A -85,B 0,C 180,E1 2572.648,E2 2572.648} C_VEL
LIN {X 0,Y 309.771,Z 718.948,A -85,B 0,C 180,E1 2570.465,E2 2570.465} C_VEL
LIN {X 0,Y 303.624,Z 714.339,A -85,B 0,C 180,E1 2566.769,E2 2566.769} C_VEL
LIN {X 0,Y 298.643,Z 710.173,A -85,B 0,C 180,E1 2563.855,E2 2563.855} C_VEL
LIN {X 0,Y 291.703,Z 704.893,A -85,B 0,C 180,E1 2560.106,E2 2560.106} C_VEL
LIN {X 0,Y 286.862,Z 700.938,A -85,B 0,C 180,E1 2557.573,E2 2557.573} C_VEL
LIN {X 0,Y 279.393,Z 695.04,A -85,B 0,C 180,E1 2553.878,E2 2553.878} C_VEL
LIN {X 0,Y 264.968,Z 683.474,A -85,B 0,C 180,E1 2546.428,E2 2546.428} C_VEL
LIN {X 0,Y 253.746,Z 669.499,A -85,B 0,C 180,E1 2537.178,E2 2537.178} C_VEL
LIN {X 0,Y 249.836,Z 657.241,A -85,B 0,C 180,E1 2529.957,E2 2529.957} C_VEL
LIN {X 0,Y 249.23,Z 652.292,A -85,B 0,C 180,E1 2527.124,E2 2527.124} C_VEL
LIN {X 0,Y 243.27,Z 673.946,A -85,B 0,C 180,E1 2526.997,E2 2526.997} C_VEL
LIN {X 0,Y 236.667,Z 691.844,A -85,B 0,C 180,E1 2526.886,E2 2526.886} C_VEL
LIN {X 0,Y 228.023,Z 710.832,A -85,B 0,C 180,E1 2526.709,E2 2526.709} C_VEL
LIN {X 0,Y 217.342,Z 729.619,A -85,B 0,C 180,E1 2526.459,E2 2526.459} C_VEL
LIN {X 0,Y 206.657,Z 745.469,A -85,B 0,C 180,E1 2526.157,E2 2526.157} C_VEL
LIN {X 0,Y 192.412,Z 763.25,A -85,B 0,C 180,E1 2525.682,E2 2525.682} C_VEL
LIN {X 0,Y 178.572,Z 777.801,A -85,B 0,C 180,E1 2525.125,E2 2525.125} C_VEL
LIN {X 0,Y 162.436,Z 792.371,A -85,B 0,C 180,E1 2524.33,E2 2524.33} C_VEL
LIN {X 0,Y 146.221,Z 804.649,A -85,B 0,C 180,E1 2523.323,E2 2523.323} C_VEL
LIN {X 0,Y 130.06,Z 815.167,A -85,B 0,C 180,E1 2522.043,E2 2522.043} C_VEL
LIN {X 0,Y 109.981,Z 826.082,A -85,B 0,C 180,E1 2519.89,E2 2519.89} C_VEL
LIN {X 0,Y 93.085,Z 833.607,A -85,B 0,C 180,E1 2517.326,E2 2517.326} C_VEL
LIN {X 0,Y 74.526,Z 840.438,A -85,B 0,C 180,E1 2513.105,E2 2513.105} C_VEL
LIN {X 0,Y 54.789,Z 845.967,A -85,B 0,C 180,E1 2505.279,E2 2505.279} C_VEL
LIN {X 0,Y 39.345,Z 849.258,A -85,B 0,C 180,E1 2492.801,E2 2492.801} C_VEL
LIN {X 0,Y 26.541,Z 851.459,A -85,B 0,C 180,E1 2463.864,E2 2463.864} C_VEL
LIN {X 0,Y 24.073,Z 851.952,A -85,B 0,C 180,E1 2430,E2 2430} C_VEL
LIN {X 0,Y 27.056,Z 851.358,A -85,B 0,C 180,E1 2393.754,E2 2393.754} C_VEL
LIN {X 0,Y 39.345,Z 849.258,A -85,B 0,C 180,E1 2367.199,E2 2367.199} C_VEL
LIN {X 0,Y 54.789,Z 845.967,A -85,B 0,C 180,E1 2354.721,E2 2354.721} C_VEL
LIN {X 0,Y 74.526,Z 840.438,A -85,B 0,C 180,E1 2346.895,E2 2346.895} C_VEL
LIN {X 0,Y 93.085,Z 833.607,A -85,B 0,C 180,E1 2342.674,E2 2342.674} C_VEL
LIN {X 0,Y 110.981,Z 825.611,A -85,B 0,C 180,E1 2339.984,E2 2339.984} C_VEL
LIN {X 0,Y 130.06,Z 815.167,A -85,B 0,C 180,E1 2337.957,E2 2337.957} C_VEL
LIN {X 0,Y 146.221,Z 804.649,A -85,B 0,C 180,E1 2336.677,E2 2336.677} C_VEL
LIN {X 0,Y 163.45,Z 791.531,A -85,B 0,C 180,E1 2335.615,E2 2335.615} C_VEL
LIN {X 0,Y 178.685,Z 777.689,A -85,B 0,C 180,E1 2334.87,E2 2334.87} C_VEL
LIN {X 0,Y 191.978,Z 763.728,A -85,B 0,C 180,E1 2334.334,E2 2334.334} C_VEL
LIN {X 0,Y 206.148,Z 746.18,A -85,B 0,C 180,E1 2333.859,E2 2333.859} C_VEL
LIN {X 0,Y 216.834,Z 730.425,A -85,B 0,C 180,E1 2333.553,E2 2333.553} C_VEL
LIN {X 0,Y 227.006,Z 712.81,A -85,B 0,C 180,E1 2333.312,E2 2333.312} C_VEL
LIN {X 0,Y 236.159,Z 693.089,A -85,B 0,C 180,E1 2333.123,E2 2333.123} C_VEL
LIN {X 0,Y 243.017,Z 674.689,A -85,B 0,C 180,E1 2333.006,E2 2333.006} C_VEL
LIN {X 0,Y 249.183,Z 652.509,A -85,B 0,C 180,E1 2332.877,E2 2332.877} C_VEL
LIN {X 0,Y 249.274,Z 652.11,A -85,B 0,C 180,E1 2332.868,E2 2332.868} C_VEL
LIN {X 0,Y 251.565,Z 664.276,A -85,B 0,C 180,E1 2325.98,E2 2325.98} C_VEL
LIN {X 0,Y 252.409,Z 666.32,A -85,B 0,C 180,E1 2324.694,E2 2324.694} C_VEL
LIN {X 0,Y 253.298,Z 670.474,A -85,B 0,C 180,E1 2322.931,E2 2322.931} C_VEL
LIN {X 0,Y 254.779,Z 681.79,A -85,B 0,C 180,E1 2319.218,E2 2319.218} C_VEL
LIN {X 0,Y 255.93,Z 684.529,A -85,B 0,C 180,E1 2317.889,E2 2317.889} C_VEL
LIN {X 0,Y 272.964,Z 699.959,A -85,B 0,C 180,E1 2307.401,E2 2307.401} C_VEL
LIN {X 0,Y 280.033,Z 705.762,A -85,B 0,C 180,E1 2303.919,E2 2303.919} C_VEL
LIN {X 0,Y 285.872,Z 710.189,A -85,B 0,C 180,E1 2300.997,E2 2300.997} C_VEL
LIN {X 0,Y 292.97,Z 715.917,A -85,B 0,C 180,E1 2297.201,E2 2297.201} C_VEL
LIN {X 0,Y 297.278,Z 719.154,A -85,B 0,C 180,E1 2294.808,E2 2294.808} C_VEL
LIN {X 0,Y 303.545,Z 724.313,A -85,B 0,C 180,E1 2291.052,E2 2291.052} C_VEL
LIN {X 0,Y 308.496,Z 727.866,A -85,B 0,C 180,E1 2288.009,E2 2288.009} C_VEL
LIN {X 0,Y 313.731,Z 732.279,A -85,B 0,C 180,E1 2284.388,E2 2284.388} C_VEL
LIN {X 0,Y 318.598,Z 735.519,A -85,B 0,C 180,E1 2280.975,E2 2280.975} C_VEL
LIN {X 0,Y 321.131,Z 737.494,A -85,B 0,C 180,E1 2278.989,E2 2278.989} C_VEL
LIN {X 0,Y 325.027,Z 740.928,A -85,B 0,C 180,E1 2275.509,E2 2275.509} C_VEL
LIN {X 0,Y 329.026,Z 743.634,A -85,B 0,C 180,E1 2271.76,E2 2271.76} C_VEL
LIN {X 0,Y 332.302,Z 745.253,A -85,B 0,C 180,E1 2268.417,E2 2268.417} C_VEL
LIN {X 0,Y 333.613,Z 746.229,A -85,B 0,C 180,E1 2266.721,E2 2266.721} C_VEL
LIN {X 0,Y 335.762,Z 748.65,A -85,B 0,C 180,E1 2263.08,E2 2263.08} C_VEL
LIN {X 0,Y 337.47,Z 750.188,A -85,B 0,C 180,E1 2259.722,E2 2259.722} C_VEL
LIN {X 0,Y 338.599,Z 751.067,A -85,B 0,C 180,E1 2256.443,E2 2256.443} C_VEL
LIN {X 0,Y 339.414,Z 751.601,A -85,B 0,C 180,E1 2253.039,E2 2253.039} C_VEL
LIN {X 0,Y 339.541,Z 751.743,A -85,B 0,C 180,E1 2249.831,E2 2249.831} C_VEL
LIN {X 0,Y 339.347,Z 751.556,A -85,B 0,C 180,E1 2246.791,E2 2246.791} C_VEL
LIN {X 0,Y 338.555,Z 751.037,A -85,B 0,C 180,E1 2243.386,E2 2243.386} C_VEL
LIN {X 0,Y 337.435,Z 750.165,A -85,B 0,C 180,E1 2240.277,E2 2240.277} C_VEL
LIN {X 0,Y 335.65,Z 748.554,A -85,B 0,C 180,E1 2236.74,E2 2236.74} C_VEL
LIN {X 0,Y 333.659,Z 746.26,A -85,B 0,C 180,E1 2233.282,E2 2233.282} C_VEL
LIN {X 0,Y 332.134,Z 745.182,A -85,B 0,C 180,E1 2231.392,E2 2231.392} C_VEL
LIN {X 0,Y 328.78,Z 743.497,A -85,B 0,C 180,E1 2228.024,E2 2228.024} C_VEL
LIN {X 0,Y 324.741,Z 740.72,A -85,B 0,C 180,E1 2224.271,E2 2224.271} C_VEL
LIN {X 0,Y 321.03,Z 737.405,A -85,B 0,C 180,E1 2220.932,E2 2220.932} C_VEL
LIN {X 0,Y 318.508,Z 735.473,A -85,B 0,C 180,E1 2218.959,E2 2218.959} C_VEL
LIN {X 0,Y 313.447,Z 732.065,A -85,B 0,C 180,E1 2215.404,E2 2215.404} C_VEL
LIN {X 0,Y 308.125,Z 727.507,A -85,B 0,C 180,E1 2211.729,E2 2211.729} C_VEL
LIN {X 0,Y 301.798,Z 722.991,A -85,B 0,C 180,E1 2207.895,E2 2207.895} C_VEL
LIN {X 0,Y 295.538,Z 717.663,A -85,B 0,C 180,E1 2204.166,E2 2204.166} C_VEL
LIN {X 0,Y 288.473,Z 712.439,A -85,B 0,C 180,E1 2200.387,E2 2200.387} C_VEL
LIN {X 0,Y 283.228,Z 708.099,A -85,B 0,C 180,E1 2197.628,E2 2197.628} C_VEL
LIN {X 0,Y 275.727,Z 702.241,A -85,B 0,C 180,E1 2193.935,E2 2193.935} C_VEL
LIN {X 0,Y 262.52,Z 691.523,A -85,B 0,C 180,E1 2186.939,E2 2186.939} C_VEL
LIN {X 0,Y 251.394,Z 677.995,A -85,B 0,C 180,E1 2177.582,E2 2177.582} C_VEL
LIN {X 0,Y 247.528,Z 664.953,A -85,B 0,C 180,E1 2169.639,E2 2169.639} C_VEL
LIN {X 0,Y 247.371,Z 663.717,A -85,B 0,C 180,E1 2168.896,E2 2168.896} C_VEL
LIN {X 0,Y 240.814,Z 683.99,A -85,B 0,C 180,E1 2168.832,E2 2168.832} C_VEL
LIN {X 0,Y 232.67,Z 703.234,A -85,B 0,C 180,E1 2168.752,E2 2168.752} C_VEL
LIN {X 0,Y 222.986,Z 721.811,A -85,B 0,C 180,E1 2168.629,E2 2168.629} C_VEL
LIN {X 0,Y 210.957,Z 740.67,A -85,B 0,C 180,E1 2168.436,E2 2168.436} C_VEL
LIN {X 0,Y 199,Z 756.377,A -85,B 0,C 180,E1 2168.2,E2 2168.2} C_VEL
LIN {X 0,Y 184.191,Z 772.945,A -85,B 0,C 180,E1 2167.841,E2 2167.841} C_VEL
LIN {X 0,Y 169.381,Z 786.85,A -85,B 0,C 180,E1 2167.398,E2 2167.398} C_VEL
LIN {X 0,Y 153.043,Z 800.088,A -85,B 0,C 180,E1 2166.777,E2 2166.777} C_VEL
LIN {X 0,Y 134.684,Z 812.445,A -85,B 0,C 180,E1 2165.875,E2 2165.875} C_VEL
LIN {X 0,Y 118.398,Z 821.733,A -85,B 0,C 180,E1 2164.815,E2 2164.815} C_VEL
LIN {X 0,Y 98.115,Z 831.355,A -85,B 0,C 180,E1 2162.97,E2 2162.97} C_VEL
LIN {X 0,Y 79.99,Z 838.176,A -85,B 0,C 180,E1 2160.518,E2 2160.518} C_VEL
LIN {X 0,Y 62.093,Z 843.583,A -85,B 0,C 180,E1 2156.683,E2 2156.683} C_VEL
LIN {X 0,Y 40.926,Z 848.258,A -85,B 0,C 180,E1 2147.744,E2 2147.744} C_VEL
LIN {X 0,Y 25.314,Z 850.564,A -85,B 0,C 180,E1 2130.334,E2 2130.334} C_VEL
LIN {X 0,Y 16.515,Z 851.535,A -85,B 0,C 180,E1 2091.3,E2 2091.3} C_VEL
LIN {X 0,Y 16.023,Z 851.696,A -85,B 0,C 180,E1 2066.422,E2 2066.422} C_VEL
LIN {X 0,Y 23.382,Z 850.805,A -85,B 0,C 180,E1 2013.899,E2 2013.899} C_VEL
LIN {X 0,Y 38.158,Z 848.715,A -85,B 0,C 180,E1 1994.193,E2 1994.193} C_VEL
LIN {X 0,Y 57.19,Z 844.875,A -85,B 0,C 180,E1 1984.789,E2 1984.789} C_VEL
LIN {X 0,Y 76.987,Z 839.187,A -85,B 0,C 180,E1 1980.001,E2 1980.001} C_VEL
LIN {X 0,Y 94.074,Z 832.965,A -85,B 0,C 180,E1 1977.491,E2 1977.491} C_VEL
LIN {X 0,Y 113.317,Z 824.4,A -85,B 0,C 180,E1 1975.587,E2 1975.587} C_VEL
LIN {X 0,Y 131.628,Z 814.308,A -85,B 0,C 180,E1 1974.302,E2 1974.302} C_VEL
LIN {X 0,Y 148.242,Z 803.502,A -85,B 0,C 180,E1 1973.433,E2 1973.433} C_VEL
LIN {X 0,Y 166.317,Z 789.524,A -85,B 0,C 180,E1 1972.707,E2 1972.707} C_VEL
LIN {X 0,Y 181.127,Z 775.954,A -85,B 0,C 180,E1 1972.243,E2 1972.243} C_VEL
LIN {X 0,Y 195.935,Z 760.122,A -85,B 0,C 180,E1 1971.872,E2 1971.872} C_VEL
LIN {X 0,Y 208.7,Z 743.814,A -85,B 0,C 180,E1 1971.606,E2 1971.606} C_VEL
LIN {X 0,Y 219.416,Z 727.771,A -85,B 0,C 180,E1 1971.423,E2 1971.423} C_VEL
LIN {X 0,Y 230.407,Z 707.95,A -85,B 0,C 180,E1 1971.275,E2 1971.275} C_VEL
LIN {X 0,Y 238.273,Z 690.369,A -85,B 0,C 180,E1 1971.187,E2 1971.187} C_VEL
LIN {X 0,Y 245.618,Z 669.802,A -85,B 0,C 180,E1 1971.124,E2 1971.124} C_VEL
LIN {X 0,Y 247.415,Z 663.661,A -85,B 0,C 180,E1 1971.06,E2 1971.06} C_VEL
LIN {X 0,Y 249.226,Z 672.466,A -85,B 0,C 180,E1 1965.846,E2 1965.846} C_VEL
LIN {X 0,Y 253.851,Z 681.964,A -85,B 0,C 180,E1 1959.732,E2 1959.732} C_VEL
LIN {X 0,Y 255.93,Z 684.529,A -85,B 0,C 180,E1 1957.889,E2 1957.889} C_VEL
LIN {X 0,Y 257.539,Z 688.329,A -85,B 0,C 180,E1 1956.133,E2 1956.133} C_VEL
LIN {X 0,Y 260.343,Z 699.023,A -85,B 0,C 180,E1 1952.417,E2 1952.417} C_VEL
LIN {X 0,Y 262.079,Z 701.587,A -85,B 0,C 180,E1 1951.127,E2 1951.127} C_VEL
LIN {X 0,Y 271.37,Z 708.918,A -85,B 0,C 180,E1 1946.21,E2 1946.21} C_VEL
LIN {X 0,Y 278.55,Z 714.565,A -85,B 0,C 180,E1 1942.668,E2 1942.668} C_VEL
LIN {X 0,Y 283.523,Z 718.611,A -85,B 0,C 180,E1 1940.086,E2 1940.086} C_VEL
LIN {X 0,Y 289.92,Z 723.519,A -85,B 0,C 180,E1 1936.678,E2 1936.678} C_VEL
LIN {X 0,Y 293.902,Z 726.679,A -85,B 0,C 180,E1 1934.42,E2 1934.42} C_VEL
LIN {X 0,Y 300.277,Z 731.766,A -85,B 0,C 180,E1 1930.625,E2 1930.625} C_VEL
LIN {X 0,Y 304.507,Z 734.83,A -85,B 0,C 180,E1 1928.015,E2 1928.015} C_VEL
LIN {X 0,Y 309.533,Z 739.055,A -85,B 0,C 180,E1 1924.563,E2 1924.563} C_VEL
LIN {X 0,Y 314.368,Z 742.313,A -85,B 0,C 180,E1 1921.2,E2 1921.2} C_VEL
LIN {X 0,Y 317.022,Z 744.313,A -85,B 0,C 180,E1 1919.14,E2 1919.14} C_VEL
LIN {X 0,Y 320.913,Z 747.759,A -85,B 0,C 180,E1 1915.662,E2 1915.662} C_VEL
LIN {X 0,Y 324.815,Z 750.434,A -85,B 0,C 180,E1 1912.057,E2 1912.057} C_VEL
LIN {X 0,Y 328.42,Z 752.254,A -85,B 0,C 180,E1 1908.458,E2 1908.458} C_VEL
LIN {X 0,Y 329.79,Z 753.292,A -85,B 0,C 180,E1 1906.695,E2 1906.695} C_VEL
LIN {X 0,Y 331.818,Z 755.58,A -85,B 0,C 180,E1 1903.238,E2 1903.238} C_VEL
LIN {X 0,Y 333.516,Z 757.135,A -85,B 0,C 180,E1 1899.839,E2 1899.839} C_VEL
LIN {X 0,Y 334.715,Z 758.07,A -85,B 0,C 180,E1 1896.345,E2 1896.345} C_VEL
LIN {X 0,Y 335.53,Z 758.597,A -85,B 0,C 180,E1 1892.904,E2 1892.904} C_VEL
LIN {X 0,Y 335.642,Z 758.723,A -85,B 0,C 180,E1 1889.659,E2 1889.659} C_VEL
LIN {X 0,Y 335.421,Z 758.52,A -85,B 0,C 180,E1 1886.411,E2 1886.411} C_VEL
LIN {X 0,Y 334.5,Z 757.909,A -85,B 0,C 180,E1 1882.961,E2 1882.961} C_VEL
LIN {X 0,Y 333.268,Z 756.953,A -85,B 0,C 180,E1 1879.63,E2 1879.63} C_VEL
LIN {X 0,Y 331.61,Z 755.39,A -85,B 0,C 180,E1 1876.398,E2 1876.398} C_VEL
LIN {X 0,Y 329.553,Z 752.966,A -85,B 0,C 180,E1 1872.885,E2 1872.885} C_VEL
LIN {X 0,Y 326.629,Z 751.42,A -85,B 0,C 180,E1 1869.763,E2 1869.763} C_VEL
LIN {X 0,Y 323.297,Z 749.474,A -85,B 0,C 180,E1 1866.488,E2 1866.488} C_VEL
LIN {X 0,Y 318.973,Z 746.138,A -85,B 0,C 180,E1 1862.563,E2 1862.563} C_VEL
LIN {X 0,Y 315.33,Z 742.864,A -85,B 0,C 180,E1 1859.515,E2 1859.515} C_VEL
LIN {X 0,Y 310.541,Z 739.812,A -85,B 0,C 180,E1 1856.149,E2 1856.149} C_VEL
LIN {X 0,Y 305.503,Z 735.756,A -85,B 0,C 180,E1 1852.664,E2 1852.664} C_VEL
LIN {X 0,Y 302.077,Z 732.977,A -85,B 0,C 180,E1 1850.445,E2 1850.445} C_VEL
LIN {X 0,Y 296.024,Z 728.5,A -85,B 0,C 180,E1 1846.833,E2 1846.833} C_VEL
LIN {X 0,Y 290.674,Z 724.028,A -85,B 0,C 180,E1 1843.725,E2 1843.725} C_VEL
LIN {X 0,Y 283.915,Z 718.936,A -85,B 0,C 180,E1 1840.111,E2 1840.111} C_VEL
LIN {X 0,Y 278.588,Z 714.587,A -85,B 0,C 180,E1 1837.326,E2 1837.326} C_VEL
LIN {X 0,Y 271.371,Z 708.916,A -85,B 0,C 180,E1 1833.79,E2 1833.79} C_VEL
LIN {X 0,Y 257.596,Z 697.541,A -85,B 0,C 180,E1 1826.002,E2 1826.002} C_VEL
LIN {X 0,Y 247.708,Z 683.943,A -85,B 0,C 180,E1 1816.401,E2 1816.401} C_VEL
LIN {X 0,Y 245.235,Z 674.981,A -85,B 0,C 180,E1 1810.715,E2 1810.715} C_VEL
LIN {X 0,Y 238.618,Z 692.624,A -85,B 0,C 180,E1 1810.712,E2 1810.712} C_VEL
LIN {X 0,Y 229.293,Z 712.607,A -85,B 0,C 180,E1 1810.685,E2 1810.685} C_VEL
LIN {X 0,Y 218.722,Z 730.763,A -85,B 0,C 180,E1 1810.638,E2 1810.638} C_VEL
LIN {X 0,Y 206.453,Z 748.468,A -85,B 0,C 180,E1 1810.547,E2 1810.547} C_VEL
LIN {X 0,Y 192.642,Z 765.023,A -85,B 0,C 180,E1 1810.416,E2 1810.416} C_VEL
LIN {X 0,Y 177.792,Z 780.206,A -85,B 0,C 180,E1 1810.221,E2 1810.221} C_VEL
LIN {X 0,Y 161.399,Z 794.301,A -85,B 0,C 180,E1 1809.947,E2 1809.947} C_VEL
LIN {X 0,Y 144.994,Z 806.285,A -85,B 0,C 180,E1 1809.572,E2 1809.572} C_VEL
LIN {X 0,Y 125.514,Z 818.228,A -85,B 0,C 180,E1 1808.972,E2 1808.972} C_VEL
LIN {X 0,Y 108.096,Z 827.018,A -85,B 0,C 180,E1 1808.234,E2 1808.234} C_VEL
LIN {X 0,Y 88.981,Z 835.011,A -85,B 0,C 180,E1 1807.071,E2 1807.071} C_VEL
LIN {X 0,Y 67.826,Z 841.816,A -85,B 0,C 180,E1 1805.037,E2 1805.037} C_VEL
LIN {X 0,Y 50.024,Z 846.126,A -85,B 0,C 180,E1 1802.067,E2 1802.067} C_VEL
LIN {X 0,Y 29.141,Z 849.658,A -85,B 0,C 180,E1 1794.268,E2 1794.268} C_VEL
LIN {X 0,Y 11.285,Z 851.196,A -85,B 0,C 180,E1 1762.879,E2 1762.879} C_VEL
LIN {X 0,Y 8.025,Z 851.458,A -85,B 0,C 180,E1 1702.843,E2 1702.843} C_VEL
LIN {X 0,Y 19.636,Z 850.605,A -85,B 0,C 180,E1 1634.657,E2 1634.657} C_VEL
LIN {X 0,Y 37.536,Z 848.396,A -85,B 0,C 180,E1 1621.593,E2 1621.593} C_VEL
LIN {X 0,Y 58.107,Z 844.401,A -85,B 0,C 180,E1 1616.371,E2 1616.371} C_VEL
LIN {X 0,Y 78.444,Z 838.609,A -85,B 0,C 180,E1 1613.808,E2 1613.808} C_VEL
LIN {X 0,Y 96.835,Z 831.921,A -85,B 0,C 180,E1 1612.395,E2 1612.395} C_VEL
LIN {X 0,Y 117.316,Z 822.581,A -85,B 0,C 180,E1 1611.346,E2 1611.346} C_VEL
LIN {X 0,Y 134.741,Z 812.827,A -85,B 0,C 180,E1 1610.718,E2 1610.718} C_VEL
LIN {X 0,Y 152.17,Z 801.334,A -85,B 0,C 180,E1 1610.256,E2 1610.256} C_VEL
LIN {X 0,Y 169.596,Z 787.504,A -85,B 0,C 180,E1 1609.907,E2 1609.907} C_VEL
LIN {X 0,Y 184.091,Z 774.07,A -85,B 0,C 180,E1 1609.689,E2 1609.689} C_VEL
LIN {X 0,Y 199.804,Z 756.773,A -85,B 0,C 180,E1 1609.512,E2 1609.512} C_VEL
LIN {X 0,Y 211.895,Z 740.993,A -85,B 0,C 180,E1 1609.408,E2 1609.408} C_VEL
LIN {X 0,Y 223.827,Z 722.463,A -85,B 0,C 180,E1 1609.337,E2 1609.337} C_VEL
LIN {X 0,Y 233.519,Z 704.068,A -85,B 0,C 180,E1 1609.302,E2 1609.302} C_VEL
LIN {X 0,Y 241.885,Z 684.569,A -85,B 0,C 180,E1 1609.291,E2 1609.291} C_VEL
LIN {X 0,Y 245.241,Z 674.98,A -85,B 0,C 180,E1 1609.277,E2 1609.277} C_VEL
LIN {X 0,Y 249.628,Z 687.82,A -85,B 0,C 180,E1 1600.952,E2 1600.952} C_VEL
LIN {X 0,Y 259.212,Z 698.911,A -85,B 0,C 180,E1 1592.938,E2 1592.938} C_VEL
LIN {X 0,Y 262.079,Z 701.587,A -85,B 0,C 180,E1 1591.127,E2 1591.127} C_VEL
LIN {X 0,Y 264.176,Z 704.683,A -85,B 0,C 180,E1 1589.64,E2 1589.64} C_VEL
LIN {X 0,Y 268.278,Z 715.817,A -85,B 0,C 180,E1 1585.83,E2 1585.83} C_VEL
LIN {X 0,Y 270.337,Z 718.38,A -85,B 0,C 180,E1 1584.59,E2 1584.59} C_VEL
LIN {X 0,Y 277.225,Z 723.634,A -85,B 0,C 180,E1 1581.145,E2 1581.145} C_VEL
LIN {X 0,Y 284.051,Z 729.165,A -85,B 0,C 180,E1 1577.496,E2 1577.496} C_VEL
LIN {X 0,Y 288.93,Z 732.844,A -85,B 0,C 180,E1 1574.829,E2 1574.829} C_VEL
LIN {X 0,Y 295.35,Z 738.068,A -85,B 0,C 180,E1 1570.998,E2 1570.998} C_VEL
LIN {X 0,Y 300.026,Z 741.418,A -85,B 0,C 180,E1 1568.16,E2 1568.16} C_VEL
LIN {X 0,Y 305.43,Z 745.951,A -85,B 0,C 180,E1 1564.437,E2 1564.437} C_VEL
LIN {X 0,Y 310.348,Z 749.224,A -85,B 0,C 180,E1 1561.028,E2 1561.028} C_VEL
LIN {X 0,Y 313.011,Z 751.333,A -85,B 0,C 180,E1 1558.95,E2 1558.95} C_VEL
LIN {X 0,Y 317.231,Z 754.968,A -85,B 0,C 180,E1 1555.181,E2 1555.181} C_VEL
LIN {X 0,Y 320.664,Z 757.271,A -85,B 0,C 180,E1 1551.972,E2 1551.972} C_VEL
LIN {X 0,Y 324.523,Z 759.193,A -85,B 0,C 180,E1 1548.13,E2 1548.13} C_VEL
LIN {X 0,Y 326.022,Z 760.656,A -85,B 0,C 180,E1 1546.022,E2 1546.022} C_VEL
LIN {X 0,Y 327.915,Z 762.693,A -85,B 0,C 180,E1 1542.682,E2 1542.682} C_VEL
LIN {X 0,Y 329.549,Z 764.162,A -85,B 0,C 180,E1 1539.077,E2 1539.077} C_VEL
LIN {X 0,Y 330.662,Z 764.991,A -85,B 0,C 180,E1 1535.901,E2 1535.901} C_VEL
LIN {X 0,Y 331.345,Z 765.445,A -85,B 0,C 180,E1 1532.421,E2 1532.421} C_VEL
LIN {X 0,Y 331.46,Z 765.534,A -85,B 0,C 180,E1 1529.482,E2 1529.482} C_VEL
LIN {X 0,Y 331.204,Z 765.329,A -85,B 0,C 180,E1 1526.192,E2 1526.192} C_VEL
LIN {X 0,Y 330.265,Z 764.694,A -85,B 0,C 180,E1 1522.87,E2 1522.87} C_VEL
LIN {X 0,Y 328.971,Z 763.694,A -85,B 0,C 180,E1 1519.493,E2 1519.493} C_VEL
LIN {X 0,Y 327.186,Z 761.992,A -85,B 0,C 180,E1 1516.03,E2 1516.03} C_VEL
LIN {X 0,Y 325.356,Z 759.776,A -85,B 0,C 180,E1 1512.842,E2 1512.842} C_VEL
LIN {X 0,Y 322.121,Z 758.08,A -85,B 0,C 180,E1 1509.467,E2 1509.467} C_VEL
LIN {X 0,Y 318.511,Z 755.891,A -85,B 0,C 180,E1 1505.965,E2 1505.965} C_VEL
LIN {X 0,Y 314.21,Z 752.467,A -85,B 0,C 180,E1 1502.111,E2 1502.111} C_VEL
LIN {X 0,Y 311.047,Z 749.626,A -85,B 0,C 180,E1 1499.461,E2 1499.461} C_VEL
LIN {X 0,Y 306.127,Z 746.473,A -85,B 0,C 180,E1 1496.037,E2 1496.037} C_VEL
LIN {X 0,Y 301.001,Z 742.339,A -85,B 0,C 180,E1 1492.533,E2 1492.533} C_VEL
LIN {X 0,Y 297.537,Z 739.569,A -85,B 0,C 180,E1 1490.295,E2 1490.295} C_VEL
LIN {X 0,Y 291.054,Z 734.698,A -85,B 0,C 180,E1 1486.439,E2 1486.439} C_VEL
LIN {X 0,Y 285.972,Z 730.505,A -85,B 0,C 180,E1 1483.518,E2 1483.518} C_VEL
LIN {X 0,Y 278.746,Z 724.965,A -85,B 0,C 180,E1 1479.664,E2 1479.664} C_VEL
LIN {X 0,Y 274.095,Z 721.201,A -85,B 0,C 180,E1 1477.253,E2 1477.253} C_VEL
LIN {X 0,Y 263.388,Z 712.742,A -85,B 0,C 180,E1 1471.834,E2 1471.834} C_VEL
LIN {X 0,Y 248.626,Z 698.47,A -85,B 0,C 180,E1 1461.454,E2 1461.454} C_VEL
LIN {X 0,Y 244.024,Z 690.133,A -85,B 0,C 180,E1 1455.434,E2 1455.434} C_VEL
LIN {X 0,Y 242.853,Z 685.984,A -85,B 0,C 180,E1 1452.571,E2 1452.571} C_VEL
LIN {X 0,Y 234.636,Z 704.902,A -85,B 0,C 180,E1 1452.628,E2 1452.628} C_VEL
LIN {X 0,Y 224.436,Z 724.008,A -85,B 0,C 180,E1 1452.68,E2 1452.68} C_VEL
LIN {X 0,Y 212.741,Z 741.856,A -85,B 0,C 180,E1 1452.727,E2 1452.727} C_VEL
LIN {X 0,Y 200.412,Z 757.783,A -85,B 0,C 180,E1 1452.756,E2 1452.756} C_VEL
LIN {X 0,Y 185.148,Z 774.391,A -85,B 0,C 180,E1 1452.777,E2 1452.777} C_VEL
LIN {X 0,Y 170.184,Z 788.158,A -85,B 0,C 180,E1 1452.775,E2 1452.775} C_VEL
LIN {X 0,Y 152.736,Z 801.827,A -85,B 0,C 180,E1 1452.742,E2 1452.742} C_VEL
LIN {X 0,Y 135.273,Z 813.209,A -85,B 0,C 180,E1 1452.674,E2 1452.674} C_VEL
LIN {X 0,Y 116.77,Z 823.415,A -85,B 0,C 180,E1 1452.549,E2 1452.549} C_VEL
LIN {X 0,Y 97.232,Z 832.084,A -85,B 0,C 180,E1 1452.346,E2 1452.346} C_VEL
LIN {X 0,Y 78.723,Z 838.706,A -85,B 0,C 180,E1 1452.054,E2 1452.054} C_VEL
LIN {X 0,Y 56.117,Z 844.824,A -85,B 0,C 180,E1 1451.501,E2 1451.501} C_VEL
LIN {X 0,Y 36.633,Z 848.39,A -85,B 0,C 180,E1 1450.718,E2 1450.718} C_VEL
LIN {X 0,Y 16.206,Z 850.638,A -85,B 0,C 180,E1 1449.216,E2 1449.216} C_VEL
LIN {X 0,Y 0.023,Z 851.241,A -85,B 0,C 180,E1 1350,E2 1350} C_VEL
LIN {X 0,Y 19.262,Z 850.367,A -85,B 0,C 180,E1 1250.477,E2 1250.477} C_VEL
LIN {X 0,Y 37.657,Z 848.237,A -85,B 0,C 180,E1 1249.231,E2 1249.231} C_VEL
LIN {X 0,Y 58.171,Z 844.386,A -85,B 0,C 180,E1 1248.438,E2 1248.438} C_VEL
LIN {X 0,Y 78.723,Z 838.705,A -85,B 0,C 180,E1 1247.946,E2 1247.946} C_VEL
LIN {X 0,Y 97.232,Z 832.084,A -85,B 0,C 180,E1 1247.654,E2 1247.654} C_VEL
LIN {X 0,Y 117.798,Z 822.886,A -85,B 0,C 180,E1 1247.442,E2 1247.442} C_VEL
LIN {X 0,Y 135.273,Z 813.209,A -85,B 0,C 180,E1 1247.326,E2 1247.326} C_VEL
LIN {X 0,Y 152.736,Z 801.827,A -85,B 0,C 180,E1 1247.258,E2 1247.258} C_VEL
LIN {X 0,Y 170.184,Z 788.158,A -85,B 0,C 180,E1 1247.225,E2 1247.225} C_VEL
LIN {X 0,Y 185.143,Z 774.396,A -85,B 0,C 180,E1 1247.222,E2 1247.222} C_VEL
LIN {X 0,Y 200.412,Z 757.782,A -85,B 0,C 180,E1 1247.245,E2 1247.245} C_VEL
LIN {X 0,Y 213.123,Z 741.324,A -85,B 0,C 180,E1 1247.275,E2 1247.275} C_VEL
LIN {X 0,Y 224.947,Z 723.115,A -85,B 0,C 180,E1 1247.322,E2 1247.322} C_VEL
LIN {X 0,Y 234.636,Z 704.902,A -85,B 0,C 180,E1 1247.373,E2 1247.373} C_VEL
LIN {X 0,Y 242.942,Z 685.803,A -85,B 0,C 180,E1 1247.412,E2 1247.412} C_VEL
LIN {X 0,Y 246.924,Z 696.11,A -85,B 0,C 180,E1 1240.373,E2 1240.373} C_VEL
LIN {X 0,Y 263.389,Z 712.74,A -85,B 0,C 180,E1 1228.166,E2 1228.166} C_VEL
LIN {X 0,Y 270.337,Z 718.38,A -85,B 0,C 180,E1 1224.59,E2 1224.59} C_VEL
LIN {X 0,Y 272.631,Z 721.462,A -85,B 0,C 180,E1 1223.164,E2 1223.164} C_VEL
LIN {X 0,Y 276.285,Z 732.367,A -85,B 0,C 180,E1 1219.418,E2 1219.418} C_VEL
LIN {X 0,Y 278.139,Z 734.741,A -85,B 0,C 180,E1 1218.183,E2 1218.183} C_VEL
LIN {X 0,Y 283.929,Z 739.044,A -85,B 0,C 180,E1 1215.056,E2 1215.056} C_VEL
LIN {X 0,Y 290.643,Z 744.536,A -85,B 0,C 180,E1 1211.075,E2 1211.075} C_VEL
LIN {X 0,Y 295.305,Z 747.859,A -85,B 0,C 180,E1 1208.25,E2 1208.25} C_VEL
LIN {X 0,Y 300.524,Z 752.263,A -85,B 0,C 180,E1 1204.674,E2 1204.674} C_VEL
LIN {X 0,Y 305.761,Z 755.788,A -85,B 0,C 180,E1 1201.068,E2 1201.068} C_VEL
LIN {X 0,Y 308.482,Z 757.934,A -85,B 0,C 180,E1 1198.964,E2 1198.964} C_VEL
LIN {X 0,Y 313.002,Z 761.785,A -85,B 0,C 180,E1 1194.905,E2 1194.905} C_VEL
LIN {X 0,Y 316.756,Z 764.233,A -85,B 0,C 180,E1 1191.412,E2 1191.412} C_VEL
LIN {X 0,Y 320.326,Z 765.948,A -85,B 0,C 180,E1 1187.859,E2 1187.859} C_VEL
LIN {X 0,Y 322.472,Z 768.379,A -85,B 0,C 180,E1 1184.362,E2 1184.362} C_VEL
LIN {X 0,Y 324.177,Z 770.077,A -85,B 0,C 180,E1 1181.024,E2 1181.024} C_VEL
LIN {X 0,Y 325.712,Z 771.272,A -85,B 0,C 180,E1 1177.408,E2 1177.408} C_VEL
LIN {X 0,Y 326.576,Z 771.877,A -85,B 0,C 180,E1 1174.214,E2 1174.214} C_VEL
LIN {X 0,Y 327.08,Z 772.173,A -85,B 0,C 180,E1 1170.876,E2 1170.876} C_VEL
LIN {X 0,Y 326.858,Z 772.084,A -85,B 0,C 180,E1 1167.546,E2 1167.546} C_VEL
LIN {X 0,Y 326.312,Z 771.695,A -85,B 0,C 180,E1 1164.642,E2 1164.642} C_VEL
LIN {X 0,Y 325.183,Z 770.894,A -85,B 0,C 180,E1 1161.157,E2 1161.157} C_VEL
LIN {X 0,Y 323.631,Z 769.563,A -85,B 0,C 180,E1 1157.873,E2 1157.873} C_VEL
LIN {X 0,Y 321.738,Z 767.545,A -85,B 0,C 180,E1 1154.314,E2 1154.314} C_VEL
LIN {X 0,Y 320.218,Z 765.92,A -85,B 0,C 180,E1 1151.994,E2 1151.994} C_VEL
LIN {X 0,Y 316.629,Z 764.159,A -85,B 0,C 180,E1 1148.513,E2 1148.513} C_VEL
LIN {X 0,Y 312.946,Z 761.756,A -85,B 0,C 180,E1 1145.056,E2 1145.056} C_VEL
LIN {X 0,Y 308.576,Z 758.037,A -85,B 0,C 180,E1 1141.133,E2 1141.133} C_VEL
LIN {X 0,Y 306.083,Z 755.983,A -85,B 0,C 180,E1 1139.146,E2 1139.146} C_VEL
LIN {X 0,Y 301.126,Z 752.722,A -85,B 0,C 180,E1 1135.748,E2 1135.748} C_VEL
LIN {X 0,Y 295.964,Z 748.49,A -85,B 0,C 180,E1 1132.216,E2 1132.216} C_VEL
LIN {X 0,Y 292.772,Z 746.008,A -85,B 0,C 180,E1 1130.193,E2 1130.193} C_VEL
LIN {X 0,Y 286.569,Z 741.347,A -85,B 0,C 180,E1 1126.512,E2 1126.512} C_VEL
LIN {X 0,Y 281.441,Z 737.096,A -85,B 0,C 180,E1 1123.552,E2 1123.552} C_VEL
LIN {X 0,Y 274.486,Z 731.813,A -85,B 0,C 180,E1 1119.859,E2 1119.859} C_VEL
LIN {X 0,Y 269.407,Z 727.682,A -85,B 0,C 180,E1 1117.21,E2 1117.21} C_VEL
LIN {X 0,Y 258.758,Z 719.258,A -85,B 0,C 180,E1 1111.689,E2 1111.689} C_VEL
LIN {X 0,Y 244.668,Z 705.223,A -85,B 0,C 180,E1 1101.064,E2 1101.064} C_VEL
LIN {X 0,Y 240.566,Z 697.013,A -85,B 0,C 180,E1 1094.921,E2 1094.921} C_VEL
LIN {X 0,Y 240.34,Z 696.494,A -85,B 0,C 180,E1 1094.476,E2 1094.476} C_VEL
LIN {X 0,Y 230.929,Z 715.613,A -85,B 0,C 180,E1 1094.611,E2 1094.611} C_VEL
LIN {X 0,Y 220.738,Z 732.714,A -85,B 0,C 180,E1 1094.751,E2 1094.751} C_VEL
LIN {X 0,Y 207.976,Z 750.631,A -85,B 0,C 180,E1 1094.919,E2 1094.919} C_VEL
LIN {X 0,Y 194.689,Z 766.236,A -85,B 0,C 180,E1 1095.1,E2 1095.1} C_VEL
LIN {X 0,Y 179.337,Z 781.645,A -85,B 0,C 180,E1 1095.312,E2 1095.312} C_VEL
LIN {X 0,Y 162.949,Z 795.413,A -85,B 0,C 180,E1 1095.565,E2 1095.565} C_VEL
LIN {X 0,Y 145.51,Z 807.886,A -85,B 0,C 180,E1 1095.853,E2 1095.853} C_VEL
LIN {X 0,Y 127.036,Z 818.84,A -85,B 0,C 180,E1 1096.221,E2 1096.221} C_VEL
LIN {X 0,Y 109.581,Z 827.483,A -85,B 0,C 180,E1 1096.658,E2 1096.658} C_VEL
LIN {X 0,Y 89.048,Z 835.769,A -85,B 0,C 180,E1 1097.373,E2 1097.373} C_VEL
LIN {X 0,Y 69.271,Z 841.845,A -85,B 0,C 180,E1 1098.475,E2 1098.475} C_VEL
LIN {X 0,Y 49.138,Z 846.497,A -85,B 0,C 180,E1 1100.612,E2 1100.612} C_VEL
LIN {X 0,Y 27.99,Z 849.57,A -85,B 0,C 180,E1 1106.743,E2 1106.743} C_VEL
LIN {X 0,Y 11.46,Z 850.788,A -85,B 0,C 180,E1 1132.358,E2 1132.358} C_VEL
LIN {X 0,Y 8.197,Z 850.983,A -85,B 0,C 180,E1 1177.006,E2 1177.006} C_VEL
LIN {X 0,Y 23.092,Z 850.036,A -85,B 0,C 180,E1 1229.991,E2 1229.991} C_VEL
LIN {X 0,Y 42.031,Z 847.694,A -85,B 0,C 180,E1 1238.082,E2 1238.082} C_VEL
LIN {X 0,Y 64.447,Z 843.135,A -85,B 0,C 180,E1 1241.147,E2 1241.147} C_VEL
LIN {X 0,Y 83.918,Z 837.454,A -85,B 0,C 180,E1 1242.392,E2 1242.392} C_VEL
LIN {X 0,Y 104.446,Z 829.778,A -85,B 0,C 180,E1 1243.19,E2 1243.19} C_VEL
LIN {X 0,Y 123.956,Z 820.471,A -85,B 0,C 180,E1 1243.71,E2 1243.71} C_VEL
LIN {X 0,Y 142.038,Z 810.104,A -85,B 0,C 180,E1 1244.085,E2 1244.085} C_VEL
LIN {X 0,Y 159.873,Z 797.792,A -85,B 0,C 180,E1 1244.387,E2 1244.387} C_VEL
LIN {X 0,Y 175.242,Z 785.247,A -85,B 0,C 180,E1 1244.625,E2 1244.625} C_VEL
LIN {X 0,Y 191.138,Z 770.093,A -85,B 0,C 180,E1 1244.852,E2 1244.852} C_VEL
LIN {X 0,Y 205.127,Z 754.148,A -85,B 0,C 180,E1 1245.042,E2 1245.042} C_VEL
LIN {X 0,Y 217.758,Z 737.235,A -85,B 0,C 180,E1 1245.209,E2 1245.209} C_VEL
LIN {X 0,Y 229.363,Z 718.447,A -85,B 0,C 180,E1 1245.367,E2 1245.367} C_VEL
LIN {X 0,Y 238.562,Z 700.372,A -85,B 0,C 180,E1 1245.497,E2 1245.497} C_VEL
LIN {X 0,Y 240.411,Z 696.389,A -85,B 0,C 180,E1 1245.5,E2 1245.5} C_VEL
LIN {X 0,Y 244.244,Z 704.628,A -85,B 0,C 180,E1 1239.399,E2 1239.399} C_VEL
LIN {X 0,Y 258.006,Z 718.708,A -85,B 0,C 180,E1 1228.729,E2 1228.729} C_VEL
LIN {X 0,Y 263.712,Z 723.285,A -85,B 0,C 180,E1 1225.617,E2 1225.617} C_VEL
LIN {X 0,Y 271.801,Z 729.452,A -85,B 0,C 180,E1 1221.575,E2 1221.575} C_VEL
LIN {X 0,Y 278.139,Z 734.741,A -85,B 0,C 180,E1 1218.183,E2 1218.183} C_VEL
LIN {X 0,Y 280.012,Z 737.065,A -85,B 0,C 180,E1 1216.96,E2 1216.96} C_VEL
LIN {X 0,Y 281.578,Z 742.441,A -85,B 0,C 180,E1 1214.982,E2 1214.982} C_VEL
LIN {X 0,Y 283.194,Z 748.217,A -85,B 0,C 180,E1 1212.788,E2 1212.788} C_VEL
LIN {X 0,Y 284.61,Z 750.021,A -85,B 0,C 180,E1 1211.76,E2 1211.76} C_VEL
LIN {X 0,Y 290.397,Z 754.173,A -85,B 0,C 180,E1 1208.296,E2 1208.296} C_VEL
LIN {X 0,Y 295.781,Z 758.706,A -85,B 0,C 180,E1 1204.603,E2 1204.603} C_VEL
LIN {X 0,Y 301.056,Z 762.244,A -85,B 0,C 180,E1 1200.982,E2 1200.982} C_VEL
LIN {X 0,Y 303.692,Z 764.365,A -85,B 0,C 180,E1 1198.889,E2 1198.889} C_VEL
LIN {X 0,Y 308.316,Z 768.267,A -85,B 0,C 180,E1 1194.794,E2 1194.794} C_VEL
LIN {X 0,Y 312.447,Z 770.898,A -85,B 0,C 180,E1 1190.897,E2 1190.897} C_VEL
LIN {X 0,Y 315.754,Z 772.462,A -85,B 0,C 180,E1 1187.649,E2 1187.649} C_VEL
LIN {X 0,Y 317.843,Z 774.964,A -85,B 0,C 180,E1 1184.017,E2 1184.017} C_VEL
LIN {X 0,Y 319.724,Z 776.752,A -85,B 0,C 180,E1 1180.45,E2 1180.45} C_VEL
LIN {X 0,Y 321.073,Z 777.776,A -85,B 0,C 180,E1 1176.976,E2 1176.976} C_VEL
LIN {X 0,Y 321.858,Z 778.335,A -85,B 0,C 180,E1 1173.919,E2 1173.919} C_VEL
LIN {X 0,Y 322.209,Z 778.586,A -85,B 0,C 180,E1 1170.178,E2 1170.178} C_VEL
LIN {X 0,Y 322.012,Z 778.437,A -85,B 0,C 180,E1 1167.152,E2 1167.152} C_VEL
LIN {X 0,Y 321.382,Z 778.008,A -85,B 0,C 180,E1 1163.928,E2 1163.928} C_VEL
LIN {X 0,Y 320.011,Z 776.967,A -85,B 0,C 180,E1 1160.287,E2 1160.287} C_VEL
LIN {X 0,Y 318.394,Z 775.491,A -85,B 0,C 180,E1 1156.933,E2 1156.933} C_VEL
LIN {X 0,Y 316.279,Z 773.141,A -85,B 0,C 180,E1 1153.27,E2 1153.27} C_VEL
LIN {X 0,Y 315.024,Z 772.162,A -85,B 0,C 180,E1 1151.585,E2 1151.585} C_VEL
LIN {X 0,Y 311.377,Z 770.296,A -85,B 0,C 180,E1 1148.094,E2 1148.094} C_VEL
LIN {X 0,Y 307.276,Z 767.498,A -85,B 0,C 180,E1 1144.308,E2 1144.308} C_VEL
LIN {X 0,Y 302.799,Z 763.494,A -85,B 0,C 180,E1 1140.311,E2 1140.311} C_VEL
LIN {X 0,Y 297.508,Z 759.973,A -85,B 0,C 180,E1 1136.554,E2 1136.554} C_VEL
LIN {X 0,Y 291.747,Z 755.428,A -85,B 0,C 180,E1 1132.645,E2 1132.645} C_VEL
LIN {X 0,Y 288.172,Z 752.538,A -85,B 0,C 180,E1 1130.328,E2 1130.328} C_VEL
LIN {X 0,Y 281.53,Z 747.553,A -85,B 0,C 180,E1 1126.411,E2 1126.411} C_VEL
LIN {X 0,Y 276.689,Z 743.524,A -85,B 0,C 180,E1 1123.63,E2 1123.63} C_VEL
LIN {X 0,Y 269.251,Z 737.853,A -85,B 0,C 180,E1 1119.681,E2 1119.681} C_VEL
LIN {X 0,Y 264.463,Z 733.975,A -85,B 0,C 180,E1 1117.208,E2 1117.208} C_VEL
LIN {X 0,Y 253.999,Z 725.688,A -85,B 0,C 180,E1 1111.557,E2 1111.557} C_VEL
LIN {X 0,Y 240.614,Z 712.017,A -85,B 0,C 180,E1 1100.781,E2 1100.781} C_VEL
LIN {X 0,Y 237.655,Z 706.57,A -85,B 0,C 180,E1 1096.421,E2 1096.421} C_VEL
LIN {X 0,Y 226.995,Z 726.017,A -85,B 0,C 180,E1 1096.663,E2 1096.663} C_VEL
LIN {X 0,Y 215.806,Z 742.886,A -85,B 0,C 180,E1 1096.92,E2 1096.92} C_VEL
LIN {X 0,Y 202.248,Z 760.124,A -85,B 0,C 180,E1 1097.241,E2 1097.241} C_VEL
LIN {X 0,Y 187.779,Z 775.516,A -85,B 0,C 180,E1 1097.62,E2 1097.62} C_VEL
LIN {X 0,Y 172.466,Z 789.448,A -85,B 0,C 180,E1 1098.057,E2 1098.057} C_VEL
LIN {X 0,Y 155.104,Z 802.762,A -85,B 0,C 180,E1 1098.632,E2 1098.632} C_VEL
LIN {X 0,Y 137.735,Z 813.972,A -85,B 0,C 180,E1 1099.321,E2 1099.321} C_VEL
LIN {X 0,Y 117.311,Z 824.889,A -85,B 0,C 180,E1 1100.362,E2 1100.362} C_VEL
LIN {X 0,Y 97.941,Z 833.216,A -85,B 0,C 180,E1 1101.725,E2 1101.725} C_VEL
LIN {X 0,Y 76.627,Z 840.423,A -85,B 0,C 180,E1 1104.026,E2 1104.026} C_VEL
LIN {X 0,Y 57.55,Z 845.195,A -85,B 0,C 180,E1 1107.621,E2 1107.621} C_VEL
LIN {X 0,Y 37.47,Z 848.747,A -85,B 0,C 180,E1 1115.863,E2 1115.863} C_VEL
LIN {X 0,Y 20.362,Z 850.447,A -85,B 0,C 180,E1 1140.592,E2 1140.592} C_VEL
LIN {X 0,Y 16.071,Z 850.765,A -85,B 0,C 180,E1 1170,E2 1170} C_VEL
LIN {X 0,Y 28.082,Z 849.798,A -85,B 0,C 180,E1 1215.404,E2 1215.404} C_VEL
LIN {X 0,Y 45.973,Z 847.417,A -85,B 0,C 180,E1 1228.602,E2 1228.602} C_VEL
LIN {X 0,Y 67.553,Z 842.894,A -85,B 0,C 180,E1 1234.534,E2 1234.534} C_VEL
LIN {X 0,Y 86.759,Z 837.213,A -85,B 0,C 180,E1 1237.211,E2 1237.211} C_VEL
LIN {X 0,Y 107.109,Z 829.533,A -85,B 0,C 180,E1 1238.982,E2 1238.982} C_VEL
LIN {X 0,Y 126.5,Z 820.232,A -85,B 0,C 180,E1 1240.144,E2 1240.144} C_VEL
LIN {X 0,Y 143.865,Z 810.248,A -85,B 0,C 180,E1 1240.939,E2 1240.939} C_VEL
LIN {X 0,Y 162.258,Z 797.555,A -85,B 0,C 180,E1 1241.612,E2 1241.612} C_VEL
LIN {X 0,Y 177.573,Z 785.01,A -85,B 0,C 180,E1 1242.093,E2 1242.093} C_VEL
LIN {X 0,Y 193.388,Z 769.88,A -85,B 0,C 180,E1 1242.531,E2 1242.531} C_VEL
LIN {X 0,Y 207.149,Z 754.18,A -85,B 0,C 180,E1 1242.875,E2 1242.875} C_VEL
LIN {X 0,Y 219.878,Z 737.109,A -85,B 0,C 180,E1 1243.173,E2 1243.173} C_VEL
LIN {X 0,Y 231.237,Z 718.746,A -85,B 0,C 180,E1 1243.431,E2 1243.431} C_VEL
LIN {X 0,Y 237.661,Z 706.569,A -85,B 0,C 180,E1 1243.573,E2 1243.573} C_VEL
LIN {X 0,Y 246.243,Z 718.893,A -85,B 0,C 180,E1 1233.744,E2 1233.744} C_VEL
LIN {X 0,Y 257.695,Z 728.642,A -85,B 0,C 180,E1 1226.315,E2 1226.315} C_VEL
LIN {X 0,Y 267.7,Z 736.503,A -85,B 0,C 180,E1 1221.151,E2 1221.151} C_VEL
LIN {X 0,Y 275.117,Z 742.437,A -85,B 0,C 180,E1 1217.203,E2 1217.203} C_VEL
LIN {X 0,Y 279.69,Z 745.962,A -85,B 0,C 180,E1 1214.668,E2 1214.668} C_VEL
LIN {X 0,Y 284.61,Z 750.021,A -85,B 0,C 180,E1 1211.76,E2 1211.76} C_VEL
LIN {X 0,Y 286.433,Z 752.659,A -85,B 0,C 180,E1 1210.34,E2 1210.34} C_VEL
LIN {X 0,Y 287.619,Z 758.78,A -85,B 0,C 180,E1 1207.958,E2 1207.958} C_VEL
LIN {X 0,Y 288.767,Z 763.031,A -85,B 0,C 180,E1 1206.023,E2 1206.023} C_VEL
LIN {X 0,Y 289.628,Z 764.054,A -85,B 0,C 180,E1 1205.293,E2 1205.293} C_VEL
LIN {X 0,Y 294.889,Z 767.767,A -85,B 0,C 180,E1 1201.697,E2 1201.697} C_VEL
LIN {X 0,Y 297.808,Z 769.763,A -85,B 0,C 180,E1 1199.572,E2 1199.572} C_VEL
LIN {X 0,Y 302.463,Z 773.873,A -85,B 0,C 180,E1 1195.45,E2 1195.45} C_VEL
LIN {X 0,Y 306.824,Z 776.782,A -85,B 0,C 180,E1 1191.406,E2 1191.406} C_VEL
LIN {X 0,Y 309.887,Z 778.311,A -85,B 0,C 180,E1 1188.433,E2 1188.433} C_VEL
LIN {X 0,Y 311.169,Z 779.274,A -85,B 0,C 180,E1 1186.797,E2 1186.797} C_VEL
LIN {X 0,Y 313.353,Z 781.702,A -85,B 0,C 180,E1 1183.094,E2 1183.094} C_VEL
LIN {X 0,Y 314.954,Z 783.161,A -85,B 0,C 180,E1 1179.686,E2 1179.686} C_VEL
LIN {X 0,Y 316.161,Z 784.089,A -85,B 0,C 180,E1 1176.355,E2 1176.355} C_VEL
LIN {X 0,Y 316.951,Z 784.606,A -85,B 0,C 180,E1 1172.712,E2 1172.712} C_VEL
LIN {X 0,Y 317.08,Z 784.737,A -85,B 0,C 180,E1 1169.819,E2 1169.819} C_VEL
LIN {X 0,Y 316.878,Z 784.561,A -85,B 0,C 180,E1 1166.925,E2 1166.925} C_VEL
LIN {X 0,Y 316.156,Z 784.083,A -85,B 0,C 180,E1 1163.463,E2 1163.463} C_VEL
LIN {X 0,Y 314.767,Z 783.025,A -85,B 0,C 180,E1 1159.901,E2 1159.901} C_VEL
LIN {X 0,Y 313.207,Z 781.566,A -85,B 0,C 180,E1 1156.712,E2 1156.712} C_VEL
LIN {X 0,Y 311.039,Z 779.113,A -85,B 0,C 180,E1 1152.991,E2 1152.991} C_VEL
LIN {X 0,Y 309.287,Z 778.033,A -85,B 0,C 180,E1 1150.943,E2 1150.943} C_VEL
LIN {X 0,Y 305.878,Z 776.221,A -85,B 0,C 180,E1 1147.718,E2 1147.718} C_VEL
LIN {X 0,Y 301.651,Z 773.245,A -85,B 0,C 180,E1 1143.843,E2 1143.843} C_VEL
LIN {X 0,Y 297.14,Z 769.117,A -85,B 0,C 180,E1 1139.835,E2 1139.835} C_VEL
LIN {X 0,Y 291.128,Z 765.214,A -85,B 0,C 180,E1 1135.721,E2 1135.721} C_VEL
LIN {X 0,Y 285.592,Z 760.634,A -85,B 0,C 180,E1 1131.954,E2 1131.954} C_VEL
LIN {X 0,Y 281.11,Z 757.364,A -85,B 0,C 180,E1 1129.235,E2 1129.235} C_VEL
LIN {X 0,Y 274.406,Z 751.971,A -85,B 0,C 180,E1 1125.261,E2 1125.261} C_VEL
LIN {X 0,Y 269.736,Z 748.397,A -85,B 0,C 180,E1 1122.698,E2 1122.698} C_VEL
LIN {X 0,Y 262.226,Z 742.33,A -85,B 0,C 180,E1 1118.691,E2 1118.691} C_VEL
LIN {X 0,Y 249.483,Z 732.294,A -85,B 0,C 180,E1 1111.655,E2 1111.655} C_VEL
LIN {X 0,Y 236.556,Z 719.06,A -85,B 0,C 180,E1 1100.783,E2 1100.783} C_VEL
LIN {X 0,Y 234.815,Z 716.417,A -85,B 0,C 180,E1 1098.427,E2 1098.427} C_VEL
LIN {X 0,Y 223.868,Z 734.648,A -85,B 0,C 180,E1 1098.769,E2 1098.769} C_VEL
LIN {X 0,Y 211.196,Z 752.055,A -85,B 0,C 180,E1 1099.186,E2 1099.186} C_VEL
LIN {X 0,Y 198.02,Z 767.434,A -85,B 0,C 180,E1 1099.656,E2 1099.656} C_VEL
LIN {X 0,Y 182.27,Z 782.991,A -85,B 0,C 180,E1 1100.281,E2 1100.281} C_VEL
LIN {X 0,Y 167.043,Z 795.733,A -85,B 0,C 180,E1 1100.976,E2 1100.976} C_VEL
LIN {X 0,Y 149.782,Z 808.073,A -85,B 0,C 180,E1 1101.897,E2 1101.897} C_VEL
LIN {X 0,Y 131.538,Z 818.906,A -85,B 0,C 180,E1 1103.114,E2 1103.114} C_VEL
LIN {X 0,Y 112.335,Z 828.41,A -85,B 0,C 180,E1 1104.792,E2 1104.792} C_VEL
LIN {X 0,Y 92.258,Z 836.299,A -85,B 0,C 180,E1 1107.294,E2 1107.294} C_VEL
LIN {X 0,Y 74.265,Z 841.874,A -85,B 0,C 180,E1 1110.729,E2 1110.729} C_VEL
LIN {X 0,Y 53.904,Z 846.631,A -85,B 0,C 180,E1 1117.681,E2 1117.681} C_VEL
LIN {X 0,Y 35.854,Z 849.373,A -85,B 0,C 180,E1 1132.158,E2 1132.158} C_VEL
LIN {X 0,Y 25.109,Z 850.415,A -85,B 0,C 180,E1 1160.835,E2 1160.835} C_VEL
LIN {X 0,Y 24.15,Z 850.526,A -85,B 0,C 180,E1 1170,E2 1170} C_VEL
LIN {X 0,Y 34.535,Z 849.532,A -85,B 0,C 180,E1 1205.97,E2 1205.97} C_VEL
LIN {X 0,Y 51.427,Z 847.063,A -85,B 0,C 180,E1 1221.047,E2 1221.047} C_VEL
LIN {X 0,Y 72.452,Z 842.38,A -85,B 0,C 180,E1 1228.825,E2 1228.825} C_VEL
LIN {X 0,Y 90.772,Z 836.8,A -85,B 0,C 180,E1 1232.476,E2 1232.476} C_VEL
LIN {X 0,Y 111.328,Z 828.849,A -85,B 0,C 180,E1 1235.104,E2 1235.104} C_VEL
LIN {X 0,Y 130.525,Z 819.449,A -85,B 0,C 180,E1 1236.81,E2 1236.81} C_VEL
LIN {X 0,Y 148.767,Z 808.748,A -85,B 0,C 180,E1 1238.043,E2 1238.043} C_VEL
LIN {X 0,Y 166.027,Z 796.526,A -85,B 0,C 180,E1 1238.974,E2 1238.974} C_VEL
LIN {X 0,Y 181.256,Z 783.882,A -85,B 0,C 180,E1 1239.675,E2 1239.675} C_VEL
LIN {X 0,Y 196.99,Z 768.57,A -85,B 0,C 180,E1 1240.307,E2 1240.307} C_VEL
LIN {X 0,Y 210.689,Z 752.685,A -85,B 0,C 180,E1 1240.797,E2 1240.797} C_VEL
LIN {X 0,Y 223.424,Z 735.299,A -85,B 0,C 180,E1 1241.216,E2 1241.216} C_VEL
LIN {X 0,Y 234.498,Z 716.993,A -85,B 0,C 180,E1 1241.563,E2 1241.563} C_VEL
LIN {X 0,Y 234.923,Z 716.334,A -85,B 0,C 180,E1 1241.526,E2 1241.526} C_VEL
LIN {X 0,Y 247.354,Z 730.684,A -85,B 0,C 180,E1 1229.664,E2 1229.664} C_VEL
LIN {X 0,Y 253.063,Z 735.2,A -85,B 0,C 180,E1 1226.16,E2 1226.16} C_VEL
LIN {X 0,Y 262.627,Z 742.695,A -85,B 0,C 180,E1 1221.1,E2 1221.1} C_VEL
LIN {X 0,Y 270.144,Z 748.687,A -85,B 0,C 180,E1 1217.093,E2 1217.093} C_VEL
LIN {X 0,Y 274.519,Z 752.067,A -85,B 0,C 180,E1 1214.662,E2 1214.662} C_VEL
LIN {X 0,Y 281.123,Z 757.368,A -85,B 0,C 180,E1 1210.768,E2 1210.768} C_VEL
LIN {X 0,Y 285.244,Z 760.298,A -85,B 0,C 180,E1 1208.282,E2 1208.282} C_VEL
LIN {X 0,Y 289.628,Z 764.054,A -85,B 0,C 180,E1 1205.293,E2 1205.293} C_VEL
LIN {X 0,Y 291.17,Z 766.331,A -85,B 0,C 180,E1 1203.859,E2 1203.859} C_VEL
LIN {X 0,Y 292.021,Z 772.695,A -85,B 0,C 180,E1 1201.043,E2 1201.043} C_VEL
LIN {X 0,Y 292.932,Z 776.075,A -85,B 0,C 180,E1 1199.187,E2 1199.187} C_VEL
LIN {X 0,Y 293.331,Z 776.569,A -85,B 0,C 180,E1 1198.767,E2 1198.767} C_VEL
LIN {X 0,Y 297.514,Z 780.117,A -85,B 0,C 180,E1 1195.052,E2 1195.052} C_VEL
LIN {X 0,Y 301.724,Z 782.887,A -85,B 0,C 180,E1 1191.174,E2 1191.174} C_VEL
LIN {X 0,Y 305.405,Z 784.673,A -85,B 0,C 180,E1 1187.529,E2 1187.529} C_VEL
LIN {X 0,Y 307.388,Z 787.064,A -85,B 0,C 180,E1 1184.12,E2 1184.12} C_VEL
LIN {X 0,Y 309.25,Z 788.837,A -85,B 0,C 180,E1 1180.431,E2 1180.431} C_VEL
LIN {X 0,Y 310.56,Z 789.837,A -85,B 0,C 180,E1 1177.027,E2 1177.027} C_VEL
LIN {X 0,Y 311.51,Z 790.499,A -85,B 0,C 180,E1 1173.496,E2 1173.496} C_VEL
LIN {X 0,Y 311.739,Z 790.681,A -85,B 0,C 180,E1 1170.184,E2 1170.184} C_VEL
LIN {X 0,Y 311.547,Z 790.537,A -85,B 0,C 180,E1 1167.241,E2 1167.241} C_VEL
LIN {X 0,Y 310.95,Z 790.121,A -85,B 0,C 180,E1 1164.279,E2 1164.279} C_VEL
LIN {X 0,Y 309.773,Z 789.259,A -85,B 0,C 180,E1 1160.713,E2 1160.713} C_VEL
LIN {X 0,Y 308.034,Z 787.692,A -85,B 0,C 180,E1 1157.058,E2 1157.058} C_VEL
LIN {X 0,Y 306.042,Z 785.508,A -85,B 0,C 180,E1 1153.487,E2 1153.487} C_VEL
LIN {X 0,Y 304.789,Z 784.386,A -85,B 0,C 180,E1 1151.842,E2 1151.842} C_VEL
LIN {X 0,Y 300.816,Z 782.354,A -85,B 0,C 180,E1 1147.992,E2 1147.992} C_VEL
LIN {X 0,Y 296.468,Z 779.328,A -85,B 0,C 180,E1 1143.997,E2 1143.997} C_VEL
LIN {X 0,Y 291.927,Z 775.194,A -85,B 0,C 180,E1 1139.997,E2 1139.997} C_VEL
LIN {X 0,Y 286.001,Z 771.319,A -85,B 0,C 180,E1 1135.928,E2 1135.928} C_VEL
LIN {X 0,Y 280.257,Z 766.598,A -85,B 0,C 180,E1 1132.021,E2 1132.021} C_VEL
LIN {X 0,Y 276.094,Z 763.54,A -85,B 0,C 180,E1 1129.49,E2 1129.49} C_VEL
LIN {X 0,Y 269.208,Z 758.049,A -85,B 0,C 180,E1 1125.417,E2 1125.417} C_VEL
LIN {X 0,Y 264.966,Z 754.752,A -85,B 0,C 180,E1 1123.062,E2 1123.062} C_VEL
LIN {X 0,Y 256.947,Z 748.341,A -85,B 0,C 180,E1 1118.777,E2 1118.777} C_VEL
LIN {X 0,Y 244.747,Z 738.733,A -85,B 0,C 180,E1 1111.788,E2 1111.788} C_VEL
LIN {X 0,Y 231.987,Z 725.782,A -85,B 0,C 180,E1 1100.485,E2 1100.485} C_VEL
LIN {X 0,Y 220.547,Z 743.134,A -85,B 0,C 180,E1 1100.952,E2 1100.952} C_VEL
LIN {X 0,Y 207.433,Z 759.866,A -85,B 0,C 180,E1 1101.524,E2 1101.524} C_VEL
LIN {X 0,Y 193.317,Z 775.047,A -85,B 0,C 180,E1 1102.213,E2 1102.213} C_VEL
LIN {X 0,Y 178.188,Z 788.969,A -85,B 0,C 180,E1 1103.042,E2 1103.042} C_VEL
LIN {X 0,Y 161.067,Z 802.289,A -85,B 0,C 180,E1 1104.146,E2 1104.146} C_VEL
LIN {X 0,Y 143.98,Z 813.488,A -85,B 0,C 180,E1 1105.478,E2 1105.478} C_VEL
LIN {X 0,Y 123.975,Z 824.413,A -85,B 0,C 180,E1 1107.486,E2 1107.486} C_VEL
LIN {X 0,Y 104.151,Z 833.14,A -85,B 0,C 180,E1 1110.233,E2 1110.233} C_VEL
LIN {X 0,Y 82.745,Z 840.497,A -85,B 0,C 180,E1 1114.748,E2 1114.748} C_VEL
LIN {X 0,Y 64.952,Z 845.142,A -85,B 0,C 180,E1 1121.038,E2 1121.038} C_VEL
LIN {X 0,Y 46.281,Z 848.666,A -85,B 0,C 180,E1 1134.317,E2 1134.317} C_VEL
LIN {X 0,Y 34.577,Z 850.039,A -85,B 0,C 180,E1 1156.625,E2 1156.625} C_VEL
LIN {X 0,Y 32.239,Z 850.287,A -85,B 0,C 180,E1 1170,E2 1170} C_VEL
LIN {X 0,Y 41.24,Z 849.321,A -85,B 0,C 180,E1 1199.005,E2 1199.005} C_VEL
LIN {X 0,Y 56.948,Z 846.824,A -85,B 0,C 180,E1 1214.609,E2 1214.609} C_VEL
LIN {X 0,Y 77.03,Z 842.139,A -85,B 0,C 180,E1 1223.585,E2 1223.585} C_VEL
LIN {X 0,Y 95.327,Z 836.395,A -85,B 0,C 180,E1 1228.164,E2 1228.164} C_VEL
LIN {X 0,Y 115.024,Z 828.604,A -85,B 0,C 180,E1 1231.393,E2 1231.393} C_VEL
LIN {X 0,Y 133.963,Z 819.21,A -85,B 0,C 180,E1 1233.587,E2 1233.587} C_VEL
LIN {X 0,Y 152.012,Z 808.504,A -85,B 0,C 180,E1 1235.185,E2 1235.185} C_VEL
LIN {X 0,Y 169.123,Z 796.289,A -85,B 0,C 180,E1 1236.396,E2 1236.396} C_VEL
LIN {X 0,Y 184.238,Z 783.645,A -85,B 0,C 180,E1 1237.303,E2 1237.303} C_VEL
LIN {X 0,Y 199.868,Z 768.334,A -85,B 0,C 180,E1 1238.118,E2 1238.118} C_VEL
LIN {X 0,Y 213.487,Z 752.451,A -85,B 0,C 180,E1 1238.746,E2 1238.746} C_VEL
LIN {X 0,Y 226.04,Z 735.223,A -85,B 0,C 180,E1 1239.275,E2 1239.275} C_VEL
LIN {X 0,Y 232.132,Z 725.647,A -85,B 0,C 180,E1 1239.475,E2 1239.475} C_VEL
LIN {X 0,Y 247.233,Z 740.719,A -85,B 0,C 180,E1 1226.647,E2 1226.647} C_VEL
LIN {X 0,Y 257.392,Z 748.743,A -85,B 0,C 180,E1 1220.977,E2 1220.977} C_VEL
LIN {X 0,Y 264.971,Z 754.755,A -85,B 0,C 180,E1 1216.938,E2 1216.938} C_VEL
LIN {X 0,Y 269.273,Z 758.104,A -85,B 0,C 180,E1 1214.544,E2 1214.544} C_VEL
LIN {X 0,Y 275.705,Z 763.257,A -85,B 0,C 180,E1 1210.735,E2 1210.735} C_VEL
LIN {X 0,Y 280.281,Z 766.612,A -85,B 0,C 180,E1 1207.985,E2 1207.985} C_VEL
LIN {X 0,Y 286.138,Z 771.414,A -85,B 0,C 180,E1 1203.992,E2 1203.992} C_VEL
LIN {X 0,Y 291.956,Z 775.211,A -85,B 0,C 180,E1 1199.976,E2 1199.976} C_VEL
LIN {X 0,Y 293.331,Z 776.569,A -85,B 0,C 180,E1 1198.767,E2 1198.767} C_VEL
LIN {X 0,Y 294.341,Z 778.72,A -85,B 0,C 180,E1 1197.323,E2 1197.323} C_VEL
LIN {X 0,Y 294.121,Z 784.663,A -85,B 0,C 180,E1 1194.496,E2 1194.496} C_VEL
LIN {X 0,Y 294.512,Z 787.458,A -85,B 0,C 180,E1 1192.732,E2 1192.732} C_VEL
LIN {X 0,Y 294.965,Z 787.902,A -85,B 0,C 180,E1 1192.205,E2 1192.205} C_VEL
LIN {X 0,Y 299.054,Z 790.07,A -85,B 0,C 180,E1 1188.317,E2 1188.317} C_VEL
LIN {X 0,Y 300.381,Z 791.148,A -85,B 0,C 180,E1 1186.578,E2 1186.578} C_VEL
LIN {X 0,Y 302.464,Z 793.431,A -85,B 0,C 180,E1 1182.796,E2 1182.796} C_VEL
LIN {X 0,Y 304.018,Z 794.828,A -85,B 0,C 180,E1 1179.45,E2 1179.45} C_VEL
LIN {X 0,Y 305.391,Z 795.866,A -85,B 0,C 180,E1 1175.637,E2 1175.637} C_VEL
LIN {X 0,Y 305.988,Z 796.272,A -85,B 0,C 180,E1 1172.435,E2 1172.435} C_VEL
LIN {X 0,Y 306.113,Z 796.377,A -85,B 0,C 180,E1 1169.626,E2 1169.626} C_VEL
LIN {X 0,Y 305.876,Z 796.166,A -85,B 0,C 180,E1 1166.627,E2 1166.627} C_VEL
LIN {X 0,Y 304.922,Z 795.534,A -85,B 0,C 180,E1 1162.842,E2 1162.842} C_VEL
LIN {X 0,Y 303.569,Z 794.483,A -85,B 0,C 180,E1 1159.563,E2 1159.563} C_VEL
LIN {X 0,Y 301.846,Z 792.834,A -85,B 0,C 180,E1 1156.007,E2 1156.007} C_VEL
LIN {X 0,Y 299.653,Z 790.326,A -85,B 0,C 180,E1 1152.324,E2 1152.324} C_VEL
LIN {X 0,Y 295.83,Z 788.437,A -85,B 0,C 180,E1 1148.592,E2 1148.592} C_VEL
LIN {X 0,Y 291.643,Z 785.62,A -85,B 0,C 180,E1 1144.806,E2 1144.806} C_VEL
LIN {X 0,Y 287.512,Z 782.082,A -85,B 0,C 180,E1 1141.094,E2 1141.094} C_VEL
LIN {X 0,Y 284.757,Z 779.96,A -85,B 0,C 180,E1 1138.93,E2 1138.93} C_VEL
LIN {X 0,Y 278.492,Z 775.567,A -85,B 0,C 180,E1 1134.689,E2 1134.689} C_VEL
LIN {X 0,Y 272.898,Z 770.857,A -85,B 0,C 180,E1 1130.938,E2 1130.938} C_VEL
LIN {X 0,Y 265.868,Z 765.69,A -85,B 0,C 180,E1 1126.833,E2 1126.833} C_VEL
LIN {X 0,Y 260.458,Z 761.229,A -85,B 0,C 180,E1 1123.691,E2 1123.691} C_VEL
LIN {X 0,Y 252.398,Z 754.972,A -85,B 0,C 180,E1 1119.425,E2 1119.425} C_VEL
LIN {X 0,Y 245.904,Z 750.002,A -85,B 0,C 180,E1 1115.824,E2 1115.824} C_VEL
LIN {X 0,Y 239.114,Z 744.515,A -85,B 0,C 180,E1 1111.46,E2 1111.46} C_VEL
LIN {X 0,Y 229.078,Z 734.896,A -85,B 0,C 180,E1 1102.61,E2 1102.61} C_VEL
LIN {X 0,Y 216.551,Z 752.218,A -85,B 0,C 180,E1 1103.25,E2 1103.25} C_VEL
LIN {X 0,Y 203.047,Z 768.08,A -85,B 0,C 180,E1 1104.005,E2 1104.005} C_VEL
LIN {X 0,Y 187.525,Z 783.408,A -85,B 0,C 180,E1 1104.989,E2 1104.989} C_VEL
LIN {X 0,Y 172.547,Z 796.052,A -85,B 0,C 180,E1 1106.084,E2 1106.084} C_VEL
LIN {X 0,Y 154.625,Z 808.912,A -85,B 0,C 180,E1 1107.643,E2 1107.643} C_VEL
LIN {X 0,Y 136.816,Z 819.515,A -85,B 0,C 180,E1 1109.584,E2 1109.584} C_VEL
LIN {X 0,Y 117.798,Z 828.978,A -85,B 0,C 180,E1 1112.298,E2 1112.298} C_VEL
LIN {X 0,Y 98.956,Z 836.491,A -85,B 0,C 180,E1 1116.069,E2 1116.069} C_VEL
LIN {X 0,Y 80.361,Z 842.446,A -85,B 0,C 180,E1 1121.711,E2 1121.711} C_VEL
LIN {X 0,Y 62.249,Z 846.738,A -85,B 0,C 180,E1 1131.214,E2 1131.214} C_VEL
LIN {X 0,Y 47.717,Z 849.213,A -85,B 0,C 180,E1 1147.071,E2 1147.071} C_VEL
LIN {X 0,Y 40.338,Z 850.048,A -85,B 0,C 180,E1 1170,E2 1170} C_VEL
LIN {X 0,Y 48.558,Z 849.082,A -85,B 0,C 180,E1 1194.318,E2 1194.318} C_VEL
LIN {X 0,Y 63.876,Z 846.433,A -85,B 0,C 180,E1 1209.923,E2 1209.923} C_VEL
LIN {X 0,Y 83.09,Z 841.625,A -85,B 0,C 180,E1 1219.296,E2 1219.296} C_VEL
LIN {X 0,Y 100.857,Z 835.817,A -85,B 0,C 180,E1 1224.379,E2 1224.379} C_VEL
LIN {X 0,Y 121.12,Z 827.472,A -85,B 0,C 180,E1 1228.239,E2 1228.239} C_VEL
LIN {X 0,Y 139.774,Z 817.88,A -85,B 0,C 180,E1 1230.772,E2 1230.772} C_VEL
LIN {X 0,Y 158.6,Z 806.237,A -85,B 0,C 180,E1 1232.732,E2 1232.732} C_VEL
LIN {X 0,Y 175.538,Z 793.674,A -85,B 0,C 180,E1 1234.149,E2 1234.149} C_VEL
LIN {X 0,Y 192.526,Z 778.751,A -85,B 0,C 180,E1 1235.342,E2 1235.342} C_VEL
LIN {X 0,Y 207.536,Z 763.043,A -85,B 0,C 180,E1 1236.255,E2 1236.255} C_VEL
LIN {X 0,Y 221.559,Z 745.661,A -85,B 0,C 180,E1 1237.013,E2 1237.013} C_VEL
LIN {X 0,Y 229.143,Z 734.845,A -85,B 0,C 180,E1 1237.372,E2 1237.372} C_VEL
LIN {X 0,Y 242.281,Z 747.022,A -85,B 0,C 180,E1 1226.442,E2 1226.442} C_VEL
LIN {X 0,Y 251.852,Z 754.501,A -85,B 0,C 180,E1 1220.875,E2 1220.875} C_VEL
LIN {X 0,Y 260.021,Z 760.92,A -85,B 0,C 180,E1 1216.521,E2 1216.521} C_VEL
LIN {X 0,Y 264.752,Z 764.742,A -85,B 0,C 180,E1 1213.854,E2 1213.854} C_VEL
LIN {X 0,Y 271.724,Z 770.094,A -85,B 0,C 180,E1 1209.75,E2 1209.75} C_VEL
LIN {X 0,Y 275.114,Z 772.718,A -85,B 0,C 180,E1 1207.621,E2 1207.621} C_VEL
LIN {X 0,Y 280.947,Z 777.412,A -85,B 0,C 180,E1 1203.637,E2 1203.637} C_VEL
LIN {X 0,Y 286.265,Z 780.836,A -85,B 0,C 180,E1 1200.004,E2 1200.004} C_VEL
LIN {X 0,Y 290.363,Z 784.61,A -85,B 0,C 180,E1 1196.372,E2 1196.372} C_VEL
LIN {X 0,Y 294.965,Z 787.902,A -85,B 0,C 180,E1 1192.205,E2 1192.205} C_VEL
LIN {X 0,Y 295.834,Z 789.519,A -85,B 0,C 180,E1 1190.74,E2 1190.74} C_VEL
LIN {X 0,Y 295.249,Z 793.75,A -85,B 0,C 180,E1 1188.259,E2 1188.259} C_VEL
LIN {X 0,Y 294.897,Z 796.92,A -85,B 0,C 180,E1 1186.039,E2 1186.039} C_VEL
LIN {X 0,Y 295.095,Z 797.309,A -85,B 0,C 180,E1 1185.499,E2 1185.499} C_VEL
LIN {X 0,Y 296.925,Z 799.224,A -85,B 0,C 180,E1 1182.05,E2 1182.05} C_VEL
LIN {X 0,Y 298.697,Z 800.724,A -85,B 0,C 180,E1 1178.082,E2 1178.082} C_VEL
LIN {X 0,Y 299.68,Z 801.405,A -85,B 0,C 180,E1 1174.976,E2 1174.976} C_VEL
LIN {X 0,Y 300.156,Z 801.753,A -85,B 0,C 180,E1 1172.1,E2 1172.1} C_VEL
LIN {X 0,Y 300.275,Z 801.798,A -85,B 0,C 180,E1 1169.046,E2 1169.046} C_VEL
LIN {X 0,Y 299.745,Z 801.476,A -85,B 0,C 180,E1 1165.217,E2 1165.217} C_VEL
LIN {X 0,Y 298.676,Z 800.709,A -85,B 0,C 180,E1 1161.918,E2 1161.918} C_VEL
LIN {X 0,Y 297.311,Z 799.587,A -85,B 0,C 180,E1 1158.752,E2 1158.752} C_VEL
LIN {X 0,Y 295.253,Z 797.504,A -85,B 0,C 180,E1 1154.779,E2 1154.779} C_VEL
LIN {X 0,Y 293.631,Z 795.741,A -85,B 0,C 180,E1 1152.154,E2 1152.154} C_VEL
LIN {X 0,Y 289.844,Z 793.796,A -85,B 0,C 180,E1 1148.552,E2 1148.552} C_VEL
LIN {X 0,Y 285.861,Z 791.125,A -85,B 0,C 180,E1 1144.916,E2 1144.916} C_VEL
LIN {X 0,Y 281.641,Z 787.513,A -85,B 0,C 180,E1 1141.131,E2 1141.131} C_VEL
LIN {X 0,Y 279.149,Z 785.549,A -85,B 0,C 180,E1 1139.191,E2 1139.191} C_VEL
LIN {X 0,Y 273.099,Z 781.373,A -85,B 0,C 180,E1 1135.073,E2 1135.073} C_VEL
LIN {X 0,Y 267.187,Z 776.413,A -85,B 0,C 180,E1 1131.092,E2 1131.092} C_VEL
LIN {X 0,Y 260.432,Z 771.486,A -85,B 0,C 180,E1 1127.144,E2 1127.144} C_VEL
LIN {X 0,Y 254.923,Z 766.903,A -85,B 0,C 180,E1 1123.948,E2 1123.948} C_VEL
LIN {X 0,Y 244.738,Z 758.864,A -85,B 0,C 180,E1 1118.372,E2 1118.372} C_VEL
LIN {X 0,Y 233.8,Z 750.508,A -85,B 0,C 180,E1 1111.434,E2 1111.434} C_VEL
LIN {X 0,Y 226.168,Z 743.609,A -85,B 0,C 180,E1 1104.805,E2 1104.805} C_VEL
LIN {X 0,Y 212.164,Z 761.389,A -85,B 0,C 180,E1 1105.679,E2 1105.679} C_VEL
LIN {X 0,Y 198.037,Z 776.578,A -85,B 0,C 180,E1 1106.669,E2 1106.669} C_VEL
LIN {X 0,Y 181.214,Z 791.817,A -85,B 0,C 180,E1 1108.02,E2 1108.02} C_VEL
LIN {X 0,Y 164.469,Z 804.628,A -85,B 0,C 180,E1 1109.621,E2 1109.621} C_VEL
LIN {X 0,Y 145.891,Z 816.534,A -85,B 0,C 180,E1 1111.809,E2 1111.809} C_VEL
LIN {X 0,Y 128.504,Z 825.82,A -85,B 0,C 180,E1 1114.439,E2 1114.439} C_VEL
LIN {X 0,Y 109.569,Z 834.193,A -85,B 0,C 180,E1 1118.302,E2 1118.302} C_VEL
LIN {X 0,Y 91.321,Z 840.563,A -85,B 0,C 180,E1 1123.73,E2 1123.73} C_VEL
LIN {X 0,Y 74.314,Z 845.296,A -85,B 0,C 180,E1 1131.765,E2 1131.765} C_VEL
LIN {X 0,Y 58.465,Z 848.469,A -85,B 0,C 180,E1 1145.768,E2 1145.768} C_VEL
LIN {X 0,Y 49.903,Z 849.631,A -85,B 0,C 180,E1 1163.096,E2 1163.096} C_VEL
LIN {X 0,Y 48.447,Z 849.808,A -85,B 0,C 180,E1 1170,E2 1170} C_VEL
LIN {X 0,Y 56.119,Z 848.843,A -85,B 0,C 180,E1 1190.875,E2 1190.875} C_VEL
LIN {X 0,Y 70.374,Z 846.192,A -85,B 0,C 180,E1 1205.627,E2 1205.627} C_VEL
LIN {X 0,Y 88.67,Z 841.384,A -85,B 0,C 180,E1 1215.266,E2 1215.266} C_VEL
LIN {X 0,Y 105.854,Z 835.576,A -85,B 0,C 180,E1 1220.762,E2 1220.762} C_VEL
LIN {X 0,Y 125.632,Z 827.232,A -85,B 0,C 180,E1 1225.056,E2 1225.056} C_VEL
LIN {X 0,Y 143.949,Z 817.639,A -85,B 0,C 180,E1 1227.928,E2 1227.928} C_VEL
LIN {X 0,Y 162.97,Z 805.673,A -85,B 0,C 180,E1 1230.221,E2 1230.221} C_VEL
LIN {X 0,Y 179.239,Z 793.436,A -85,B 0,C 180,E1 1231.806,E2 1231.806} C_VEL
LIN {X 0,Y 196.055,Z 778.509,A -85,B 0,C 180,E1 1233.183,E2 1233.183} C_VEL
LIN {X 0,Y 210.93,Z 762.803,A -85,B 0,C 180,E1 1234.239,E2 1234.239} C_VEL
LIN {X 0,Y 224.839,Z 745.419,A -85,B 0,C 180,E1 1235.116,E2 1235.116} C_VEL
LIN {X 0,Y 226.22,Z 743.56,A -85,B 0,C 180,E1 1235.187,E2 1235.187} C_VEL
LIN {X 0,Y 237.175,Z 753.179,A -85,B 0,C 180,E1 1226.203,E2 1226.203} C_VEL
LIN {X 0,Y 246.254,Z 760.187,A -85,B 0,C 180,E1 1220.715,E2 1220.715} C_VEL
LIN {X 0,Y 254.919,Z 766.901,A -85,B 0,C 180,E1 1216.051,E2 1216.051} C_VEL
LIN {X 0,Y 260.812,Z 771.787,A -85,B 0,C 180,E1 1212.622,E2 1212.622} C_VEL
LIN {X 0,Y 267.761,Z 776.766,A -85,B 0,C 180,E1 1208.578,E2 1208.578} C_VEL
LIN {X 0,Y 273.855,Z 781.946,A -85,B 0,C 180,E1 1204.42,E2 1204.42} C_VEL
LIN {X 0,Y 279.213,Z 785.58,A -85,B 0,C 180,E1 1200.771,E2 1200.771} C_VEL
LIN {X 0,Y 281.73,Z 787.586,A -85,B 0,C 180,E1 1198.791,E2 1198.791} C_VEL
LIN {X 0,Y 285.908,Z 791.142,A -85,B 0,C 180,E1 1195.033,E2 1195.033} C_VEL
LIN {X 0,Y 289.614,Z 793.661,A -85,B 0,C 180,E1 1191.678,E2 1191.678} C_VEL
LIN {X 0,Y 293.626,Z 795.73,A -85,B 0,C 180,E1 1187.846,E2 1187.846} C_VEL
LIN {X 0,Y 295.095,Z 797.309,A -85,B 0,C 180,E1 1185.499,E2 1185.499} C_VEL
LIN {X 0,Y 295.145,Z 798.966,A -85,B 0,C 180,E1 1184.022,E2 1184.022} C_VEL
LIN {X 0,Y 293.142,Z 803.342,A -85,B 0,C 180,E1 1181.232,E2 1181.232} C_VEL
LIN {X 0,Y 292.284,Z 805.495,A -85,B 0,C 180,E1 1179.313,E2 1179.313} C_VEL
LIN {X 0,Y 292.365,Z 805.732,A -85,B 0,C 180,E1 1178.767,E2 1178.767} C_VEL
LIN {X 0,Y 293.468,Z 806.486,A -85,B 0,C 180,E1 1175.278,E2 1175.278} C_VEL
LIN {X 0,Y 293.988,Z 806.848,A -85,B 0,C 180,E1 1172.339,E2 1172.339} C_VEL
LIN {X 0,Y 294.105,Z 806.941,A -85,B 0,C 180,E1 1169.61,E2 1169.61} C_VEL
LIN {X 0,Y 293.854,Z 806.725,A -85,B 0,C 180,E1 1166.489,E2 1166.489} C_VEL
LIN {X 0,Y 292.922,Z 806.136,A -85,B 0,C 180,E1 1162.745,E2 1162.745} C_VEL
LIN {X 0,Y 291.473,Z 804.992,A -85,B 0,C 180,E1 1159.325,E2 1159.325} C_VEL
LIN {X 0,Y 289.811,Z 803.371,A -85,B 0,C 180,E1 1156.025,E2 1156.025} C_VEL
LIN {X 0,Y 287.593,Z 800.974,A -85,B 0,C 180,E1 1152.247,E2 1152.247} C_VEL
LIN {X 0,Y 283.86,Z 799.039,A -85,B 0,C 180,E1 1148.728,E2 1148.728} C_VEL
LIN {X 0,Y 279.612,Z 796.193,A -85,B 0,C 180,E1 1144.817,E2 1144.817} C_VEL
LIN {X 0,Y 275.029,Z 792.185,A -85,B 0,C 180,E1 1140.726,E2 1140.726} C_VEL
LIN {X 0,Y 270.657,Z 789.223,A -85,B 0,C 180,E1 1137.613,E2 1137.613} C_VEL
LIN {X 0,Y 264.666,Z 784.648,A -85,B 0,C 180,E1 1133.557,E2 1133.557} C_VEL
LIN {X 0,Y 260.482,Z 781.228,A -85,B 0,C 180,E1 1130.819,E2 1130.819} C_VEL
LIN {X 0,Y 252.863,Z 775.42,A -85,B 0,C 180,E1 1126.335,E2 1126.335} C_VEL
LIN {X 0,Y 248.38,Z 771.801,A -85,B 0,C 180,E1 1123.802,E2 1123.802} C_VEL
LIN {X 0,Y 237.594,Z 763.485,A -85,B 0,C 180,E1 1117.709,E2 1117.709} C_VEL
LIN {X 0,Y 228.621,Z 756.569,A -85,B 0,C 180,E1 1111.64,E2 1111.64} C_VEL
LIN {X 0,Y 223.21,Z 752.033,A -85,B 0,C 180,E1 1107.079,E2 1107.079} C_VEL
LIN {X 0,Y 209.658,Z 768.146,A -85,B 0,C 180,E1 1108.087,E2 1108.087} C_VEL
LIN {X 0,Y 194.95,Z 782.935,A -85,B 0,C 180,E1 1109.323,E2 1109.323} C_VEL
LIN {X 0,Y 179.332,Z 796.372,A -85,B 0,C 180,E1 1110.841,E2 1110.841} C_VEL
LIN {X 0,Y 161.887,Z 809.056,A -85,B 0,C 180,E1 1112.865,E2 1112.865} C_VEL
LIN {X 0,Y 144.648,Z 819.58,A -85,B 0,C 180,E1 1115.35,E2 1115.35} C_VEL
LIN {X 0,Y 125.703,Z 829.255,A -85,B 0,C 180,E1 1118.902,E2 1118.902} C_VEL
LIN {X 0,Y 107.658,Z 836.683,A -85,B 0,C 180,E1 1123.582,E2 1123.582} C_VEL
LIN {X 0,Y 89.646,Z 842.673,A -85,B 0,C 180,E1 1130.526,E2 1130.526} C_VEL
LIN {X 0,Y 74.342,Z 846.565,A -85,B 0,C 180,E1 1140.158,E2 1140.158} C_VEL
LIN {X 0,Y 62.275,Z 848.868,A -85,B 0,C 180,E1 1154.274,E2 1154.274} C_VEL
LIN {X 0,Y 56.565,Z 849.568,A -85,B 0,C 180,E1 1170,E2 1170} C_VEL
LIN {X 0,Y 63.836,Z 848.604,A -85,B 0,C 180,E1 1188.255,E2 1188.255} C_VEL
LIN {X 0,Y 77.2,Z 845.948,A -85,B 0,C 180,E1 1202.073,E2 1202.073} C_VEL
LIN {X 0,Y 94.637,Z 841.144,A -85,B 0,C 180,E1 1211.727,E2 1211.727} C_VEL
LIN {X 0,Y 111.232,Z 835.336,A -85,B 0,C 180,E1 1217.483,E2 1217.483} C_VEL
LIN {X 0,Y 130.504,Z 826.99,A -85,B 0,C 180,E1 1222.103,E2 1222.103} C_VEL
LIN {X 0,Y 148.456,Z 817.397,A -85,B 0,C 180,E1 1225.251,E2 1225.251} C_VEL
LIN {X 0,Y 166.718,Z 805.749,A -85,B 0,C 180,E1 1227.736,E2 1227.736} C_VEL
LIN {X 0,Y 183.704,Z 792.799,A -85,B 0,C 180,E1 1229.609,E2 1229.609} C_VEL
LIN {X 0,Y 199.852,Z 778.266,A -85,B 0,C 180,E1 1231.104,E2 1231.104} C_VEL
LIN {X 0,Y 214.575,Z 762.564,A -85,B 0,C 180,E1 1232.291,E2 1232.291} C_VEL
LIN {X 0,Y 223.315,Z 751.931,A -85,B 0,C 180,E1 1232.913,E2 1232.913} C_VEL
LIN {X 0,Y 231.945,Z 759.213,A -85,B 0,C 180,E1 1225.933,E2 1225.933} C_VEL
LIN {X 0,Y 240.56,Z 765.765,A -85,B 0,C 180,E1 1220.528,E2 1220.528} C_VEL
LIN {X 0,Y 250.824,Z 773.623,A -85,B 0,C 180,E1 1214.874,E2 1214.874} C_VEL
LIN {X 0,Y 258.03,Z 779.521,A -85,B 0,C 180,E1 1210.6,E2 1210.6} C_VEL
LIN {X 0,Y 262.838,Z 783.035,A -85,B 0,C 180,E1 1207.718,E2 1207.718} C_VEL
LIN {X 0,Y 268.728,Z 787.835,A -85,B 0,C 180,E1 1203.667,E2 1203.667} C_VEL
LIN {X 0,Y 274.197,Z 791.416,A -85,B 0,C 180,E1 1199.971,E2 1199.971} C_VEL
LIN {X 0,Y 278.176,Z 795.032,A -85,B 0,C 180,E1 1196.467,E2 1196.467} C_VEL
LIN {X 0,Y 282.063,Z 797.9,A -85,B 0,C 180,E1 1192.949,E2 1192.949} C_VEL
LIN {X 0,Y 286.639,Z 800.516,A -85,B 0,C 180,E1 1188.718,E2 1188.718} C_VEL
LIN {X 0,Y 288.325,Z 801.648,A -85,B 0,C 180,E1 1186.728,E2 1186.728} C_VEL
LIN {X 0,Y 290.378,Z 803.916,A -85,B 0,C 180,E1 1182.933,E2 1182.933} C_VEL
LIN {X 0,Y 292.152,Z 805.541,A -85,B 0,C 180,E1 1179.256,E2 1179.256} C_VEL
LIN {X 0,Y 292.365,Z 805.732,A -85,B 0,C 180,E1 1178.767,E2 1178.767} C_VEL
LIN {X 0,Y 292.12,Z 806.665,A -85,B 0,C 180,E1 1177.365,E2 1177.365} C_VEL
LIN {X 0,Y 289.599,Z 809.669,A -85,B 0,C 180,E1 1174.829,E2 1174.829} C_VEL
LIN {X 0,Y 287.88,Z 811.474,A -85,B 0,C 180,E1 1172.881,E2 1172.881} C_VEL
LIN {X 0,Y 287.673,Z 811.745,A -85,B 0,C 180,E1 1171.881,E2 1171.881} C_VEL
LIN {X 0,Y 287.779,Z 811.773,A -85,B 0,C 180,E1 1168.606,E2 1168.606} C_VEL
LIN {X 0,Y 287.104,Z 811.347,A -85,B 0,C 180,E1 1164.741,E2 1164.741} C_VEL
LIN {X 0,Y 286.036,Z 810.587,A -85,B 0,C 180,E1 1161.502,E2 1161.502} C_VEL
LIN {X 0,Y 284.63,Z 809.418,A -85,B 0,C 180,E1 1158.244,E2 1158.244} C_VEL
LIN {X 0,Y 282.448,Z 807.127,A -85,B 0,C 180,E1 1154.183,E2 1154.183} C_VEL
LIN {X 0,Y 281.167,Z 805.854,A -85,B 0,C 180,E1 1152.193,E2 1152.193} C_VEL
LIN {X 0,Y 277.392,Z 803.866,A -85,B 0,C 180,E1 1148.651,E2 1148.651} C_VEL
LIN {X 0,Y 273.019,Z 800.892,A -85,B 0,C 180,E1 1144.63,E2 1144.63} C_VEL
LIN {X 0,Y 268.115,Z 796.511,A -85,B 0,C 180,E1 1140.266,E2 1140.266} C_VEL
LIN {X 0,Y 262.133,Z 792.551,A -85,B 0,C 180,E1 1136.232,E2 1136.232} C_VEL
LIN {X 0,Y 256.326,Z 787.76,A -85,B 0,C 180,E1 1132.237,E2 1132.237} C_VEL
LIN {X 0,Y 249.469,Z 782.741,A -85,B 0,C 180,E1 1128.18,E2 1128.18} C_VEL
LIN {X 0,Y 242.948,Z 777.343,A -85,B 0,C 180,E1 1124.38,E2 1124.38} C_VEL
LIN {X 0,Y 231.757,Z 768.925,A -85,B 0,C 180,E1 1117.863,E2 1117.863} C_VEL
LIN {X 0,Y 222.942,Z 762.23,A -85,B 0,C 180,E1 1111.634,E2 1111.634} C_VEL
LIN {X 0,Y 220.164,Z 760.332,A -85,B 0,C 180,E1 1109.449,E2 1109.449} C_VEL
LIN {X 0,Y 206.322,Z 775.609,A -85,B 0,C 180,E1 1110.666,E2 1110.666} C_VEL
LIN {X 0,Y 190.372,Z 790.525,A -85,B 0,C 180,E1 1112.267,E2 1112.267} C_VEL
LIN {X 0,Y 174.078,Z 803.451,A -85,B 0,C 180,E1 1114.201,E2 1114.201} C_VEL
LIN {X 0,Y 157.016,Z 814.946,A -85,B 0,C 180,E1 1116.647,E2 1116.647} C_VEL
LIN {X 0,Y 139.355,Z 824.873,A -85,B 0,C 180,E1 1119.853,E2 1119.853} C_VEL
LIN {X 0,Y 122.207,Z 832.935,A -85,B 0,C 180,E1 1123.949,E2 1123.949} C_VEL
LIN {X 0,Y 104.195,Z 839.805,A -85,B 0,C 180,E1 1129.99,E2 1129.99} C_VEL
LIN {X 0,Y 88.226,Z 844.7,A -85,B 0,C 180,E1 1138.148,E2 1138.148} C_VEL
LIN {X 0,Y 74.268,Z 847.897,A -85,B 0,C 180,E1 1150.332,E2 1150.332} C_VEL
LIN {X 0,Y 66.115,Z 849.153,A -85,B 0,C 180,E1 1164.794,E2 1164.794} C_VEL
LIN {X 0,Y 64.691,Z 849.328,A -85,B 0,C 180,E1 1170,E2 1170} C_VEL
LIN {X 0,Y 72.16,Z 848.272,A -85,B 0,C 180,E1 1186.916,E2 1186.916} C_VEL
LIN {X 0,Y 85.188,Z 845.468,A -85,B 0,C 180,E1 1199.777,E2 1199.777} C_VEL
LIN {X 0,Y 101.735,Z 840.629,A -85,B 0,C 180,E1 1208.975,E2 1208.975} C_VEL
LIN {X 0,Y 117.812,Z 834.758,A -85,B 0,C 180,E1 1214.781,E2 1214.781} C_VEL
LIN {X 0,Y 136.609,Z 826.286,A -85,B 0,C 180,E1 1219.567,E2 1219.567} C_VEL
LIN {X 0,Y 153.817,Z 816.83,A -85,B 0,C 180,E1 1222.829,E2 1222.829} C_VEL
LIN {X 0,Y 172.169,Z 804.831,A -85,B 0,C 180,E1 1225.551,E2 1225.551} C_VEL
LIN {X 0,Y 188.447,Z 792.144,A -85,B 0,C 180,E1 1227.521,E2 1227.521} C_VEL
LIN {X 0,Y 204.984,Z 776.947,A -85,B 0,C 180,E1 1229.209,E2 1229.209} C_VEL
LIN {X 0,Y 218.73,Z 762.009,A -85,B 0,C 180,E1 1230.432,E2 1230.432} C_VEL
LIN {X 0,Y 220.344,Z 760.212,A -85,B 0,C 180,E1 1230.521,E2 1230.521} C_VEL
LIN {X 0,Y 226.59,Z 765.111,A -85,B 0,C 180,E1 1225.602,E2 1225.602} C_VEL
LIN {X 0,Y 234.718,Z 771.163,A -85,B 0,C 180,E1 1220.302,E2 1220.302} C_VEL
LIN {X 0,Y 245.055,Z 779.021,A -85,B 0,C 180,E1 1214.456,E2 1214.456} C_VEL
LIN {X 0,Y 252.331,Z 784.879,A -85,B 0,C 180,E1 1210.135,E2 1210.135} C_VEL
LIN {X 0,Y 256.422,Z 787.834,A -85,B 0,C 180,E1 1207.691,E2 1207.691} C_VEL
LIN {X 0,Y 262.137,Z 792.545,A -85,B 0,C 180,E1 1203.769,E2 1203.769} C_VEL
LIN {X 0,Y 268.159,Z 796.536,A -85,B 0,C 180,E1 1199.711,E2 1199.711} C_VEL
LIN {X 0,Y 272.992,Z 800.845,A -85,B 0,C 180,E1 1195.373,E2 1195.373} C_VEL
LIN {X 0,Y 277.657,Z 804.016,A -85,B 0,C 180,E1 1191.106,E2 1191.106} C_VEL
LIN {X 0,Y 280.892,Z 805.685,A -85,B 0,C 180,E1 1188.04,E2 1188.04} C_VEL
LIN {X 0,Y 282.2,Z 806.804,A -85,B 0,C 180,E1 1186.27,E2 1186.27} C_VEL
LIN {X 0,Y 284.217,Z 808.995,A -85,B 0,C 180,E1 1182.598,E2 1182.598} C_VEL
LIN {X 0,Y 286.015,Z 810.577,A -85,B 0,C 180,E1 1178.645,E2 1178.645} C_VEL
LIN {X 0,Y 287.116,Z 811.339,A -85,B 0,C 180,E1 1175.195,E2 1175.195} C_VEL
LIN {X 0,Y 287.641,Z 811.716,A -85,B 0,C 180,E1 1172.191,E2 1172.191} C_VEL
LIN {X 0,Y 287.673,Z 811.745,A -85,B 0,C 180,E1 1171.881,E2 1171.881} C_VEL
LIN {X 0,Y 286.99,Z 812.435,A -85,B 0,C 180,E1 1170.346,E2 1170.346} C_VEL
LIN {X 0,Y 283.886,Z 814.575,A -85,B 0,C 180,E1 1167.988,E2 1167.988} C_VEL
LIN {X 0,Y 281.029,Z 815.979,A -85,B 0,C 180,E1 1165.675,E2 1165.675} C_VEL
LIN {X 0,Y 280.582,Z 815.959,A -85,B 0,C 180,E1 1164.877,E2 1164.877} C_VEL
LIN {X 0,Y 279.479,Z 815.161,A -85,B 0,C 180,E1 1161.566,E2 1161.566} C_VEL
LIN {X 0,Y 277.999,Z 813.916,A -85,B 0,C 180,E1 1158.17,E2 1158.17} C_VEL
LIN {X 0,Y 276.053,Z 811.914,A -85,B 0,C 180,E1 1154.412,E2 1154.412} C_VEL
LIN {X 0,Y 274.545,Z 810.44,A -85,B 0,C 180,E1 1152.187,E2 1152.187} C_VEL
LIN {X 0,Y 270.401,Z 808.21,A -85,B 0,C 180,E1 1148.299,E2 1148.299} C_VEL
LIN {X 0,Y 265.73,Z 804.902,A -85,B 0,C 180,E1 1144.034,E2 1144.034} C_VEL
LIN {X 0,Y 261.296,Z 800.989,A -85,B 0,C 180,E1 1140.17,E2 1140.17} C_VEL
LIN {X 0,Y 254.882,Z 796.631,A -85,B 0,C 180,E1 1135.841,E2 1135.841} C_VEL
LIN {X 0,Y 248.992,Z 791.713,A -85,B 0,C 180,E1 1131.801,E2 1131.801} C_VEL
LIN {X 0,Y 241.51,Z 786.207,A -85,B 0,C 180,E1 1127.45,E2 1127.45} C_VEL
LIN {X 0,Y 236.046,Z 781.786,A -85,B 0,C 180,E1 1124.288,E2 1124.288} C_VEL
LIN {X 0,Y 225.732,Z 774.186,A -85,B 0,C 180,E1 1117.985,E2 1117.985} C_VEL
LIN {X 0,Y 217.463,Z 767.995,A -85,B 0,C 180,E1 1111.886,E2 1111.886} C_VEL
LIN {X 0,Y 203.405,Z 782.461,A -85,B 0,C 180,E1 1113.319,E2 1113.319} C_VEL
LIN {X 0,Y 188.203,Z 795.898,A -85,B 0,C 180,E1 1115.103,E2 1115.103} C_VEL
LIN {X 0,Y 171.303,Z 808.579,A -85,B 0,C 180,E1 1117.46,E2 1117.46} C_VEL
LIN {X 0,Y 154.697,Z 819.102,A -85,B 0,C 180,E1 1120.302,E2 1120.302} C_VEL
LIN {X 0,Y 136.746,Z 828.696,A -85,B 0,C 180,E1 1124.231,E2 1124.231} C_VEL
LIN {X 0,Y 120.414,Z 835.865,A -85,B 0,C 180,E1 1129.008,E2 1129.008} C_VEL
LIN {X 0,Y 104.383,Z 841.724,A -85,B 0,C 180,E1 1135.589,E2 1135.589} C_VEL
LIN {X 0,Y 89.601,Z 845.934,A -85,B 0,C 180,E1 1144.911,E2 1144.911} C_VEL
LIN {X 0,Y 78.653,Z 848.291,A -85,B 0,C 180,E1 1156.773,E2 1156.773} C_VEL
LIN {X 0,Y 72.824,Z 849.088,A -85,B 0,C 180,E1 1170,E2 1170} C_VEL
LIN {X 0,Y 80.037,Z 848.033,A -85,B 0,C 180,E1 1185.209,E2 1185.209} C_VEL
LIN {X 0,Y 92.202,Z 845.279,A -85,B 0,C 180,E1 1197.093,E2 1197.093} C_VEL
LIN {X 0,Y 107.467,Z 840.663,A -85,B 0,C 180,E1 1205.882,E2 1205.882} C_VEL
LIN {X 0,Y 122.932,Z 834.855,A -85,B 0,C 180,E1 1211.83,E2 1211.83} C_VEL
LIN {X 0,Y 141.172,Z 826.501,A -85,B 0,C 180,E1 1216.843,E2 1216.843} C_VEL
LIN {X 0,Y 158.355,Z 816.913,A -85,B 0,C 180,E1 1220.38,E2 1220.38} C_VEL
LIN {X 0,Y 175.978,Z 805.263,A -85,B 0,C 180,E1 1223.235,E2 1223.235} C_VEL
LIN {X 0,Y 191.993,Z 792.712,A -85,B 0,C 180,E1 1225.367,E2 1225.367} C_VEL
LIN {X 0,Y 207.228,Z 778.744,A -85,B 0,C 180,E1 1227.089,E2 1227.089} C_VEL
LIN {X 0,Y 217.484,Z 768.006,A -85,B 0,C 180,E1 1228.098,E2 1228.098} C_VEL
LIN {X 0,Y 228.389,Z 776.104,A -85,B 0,C 180,E1 1220.288,E2 1220.288} C_VEL
LIN {X 0,Y 238.644,Z 783.733,A -85,B 0,C 180,E1 1214.257,E2 1214.257} C_VEL
LIN {X 0,Y 245.898,Z 789.605,A -85,B 0,C 180,E1 1209.973,E2 1209.973} C_VEL
LIN {X 0,Y 250.235,Z 792.76,A -85,B 0,C 180,E1 1207.353,E2 1207.353} C_VEL
LIN {X 0,Y 256.093,Z 797.544,A -85,B 0,C 180,E1 1203.354,E2 1203.354} C_VEL
LIN {X 0,Y 262.15,Z 801.647,A -85,B 0,C 180,E1 1199.168,E2 1199.168} C_VEL
LIN {X 0,Y 267.015,Z 805.883,A -85,B 0,C 180,E1 1194.795,E2 1194.795} C_VEL
LIN {X 0,Y 271.494,Z 808.877,A -85,B 0,C 180,E1 1190.704,E2 1190.704} C_VEL
LIN {X 0,Y 275.21,Z 810.821,A -85,B 0,C 180,E1 1187.114,E2 1187.114} C_VEL
LIN {X 0,Y 277.304,Z 813.211,A -85,B 0,C 180,E1 1183.271,E2 1183.271} C_VEL
LIN {X 0,Y 279.204,Z 814.944,A -85,B 0,C 180,E1 1179.273,E2 1179.273} C_VEL
LIN {X 0,Y 280.468,Z 815.859,A -85,B 0,C 180,E1 1175.523,E2 1175.523} C_VEL
LIN {X 0,Y 281.065,Z 816.275,A -85,B 0,C 180,E1 1172.447,E2 1172.447} C_VEL
LIN {X 0,Y 281.194,Z 816.384,A -85,B 0,C 180,E1 1169.593,E2 1169.593} C_VEL
LIN {X 0,Y 280.937,Z 816.162,A -85,B 0,C 180,E1 1166.531,E2 1166.531} C_VEL
LIN {X 0,Y 280.582,Z 815.959,A -85,B 0,C 180,E1 1164.877,E2 1164.877} C_VEL
LIN {X 0,Y 279.364,Z 816.189,A -85,B 0,C 180,E1 1163.424,E2 1163.424} C_VEL
LIN {X 0,Y 275.142,Z 817.652,A -85,B 0,C 180,E1 1160.925,E2 1160.925} C_VEL
LIN {X 0,Y 271.848,Z 818.255,A -85,B 0,C 180,E1 1158.797,E2 1158.797} C_VEL
LIN {X 0,Y 271.021,Z 817.966,A -85,B 0,C 180,E1 1157.747,E2 1157.747} C_VEL
LIN {X 0,Y 268.818,Z 815.604,A -85,B 0,C 180,E1 1153.58,E2 1153.58} C_VEL
LIN {X 0,Y 267.225,Z 814.504,A -85,B 0,C 180,E1 1151.682,E2 1151.682} C_VEL
LIN {X 0,Y 262.776,Z 811.953,A -85,B 0,C 180,E1 1147.575,E2 1147.575} C_VEL
LIN {X 0,Y 257.818,Z 808.202,A -85,B 0,C 180,E1 1143.093,E2 1143.093} C_VEL
LIN {X 0,Y 254.477,Z 805.288,A -85,B 0,C 180,E1 1140.237,E2 1140.237} C_VEL
LIN {X 0,Y 248.144,Z 800.971,A -85,B 0,C 180,E1 1135.94,E2 1135.94} C_VEL
LIN {X 0,Y 242.324,Z 796.121,A -85,B 0,C 180,E1 1131.985,E2 1131.985} C_VEL
LIN {X 0,Y 234.594,Z 790.37,A -85,B 0,C 180,E1 1127.485,E2 1127.485} C_VEL
LIN {X 0,Y 229.593,Z 786.47,A -85,B 0,C 180,E1 1124.499,E2 1124.499} C_VEL
LIN {X 0,Y 219.696,Z 779.358,A -85,B 0,C 180,E1 1118.222,E2 1118.222} C_VEL
LIN {X 0,Y 214.463,Z 775.735,A -85,B 0,C 180,E1 1114.453,E2 1114.453} C_VEL
LIN {X 0,Y 199.535,Z 790.043,A -85,B 0,C 180,E1 1116.222,E2 1116.222} C_VEL
LIN {X 0,Y 183.746,Z 802.979,A -85,B 0,C 180,E1 1118.413,E2 1118.413} C_VEL
LIN {X 0,Y 166.717,Z 814.817,A -85,B 0,C 180,E1 1121.254,E2 1121.254} C_VEL
LIN {X 0,Y 150.387,Z 824.396,A -85,B 0,C 180,E1 1124.653,E2 1124.653} C_VEL
LIN {X 0,Y 134.126,Z 832.446,A -85,B 0,C 180,E1 1129.005,E2 1129.005} C_VEL
LIN {X 0,Y 117.264,Z 839.319,A -85,B 0,C 180,E1 1135.162,E2 1135.162} C_VEL
LIN {X 0,Y 102.183,Z 844.316,A -85,B 0,C 180,E1 1143.25,E2 1143.25} C_VEL
LIN {X 0,Y 89.395,Z 847.512,A -85,B 0,C 180,E1 1154.429,E2 1154.429} C_VEL
LIN {X 0,Y 82.085,Z 848.706,A -85,B 0,C 180,E1 1166.576,E2 1166.576} C_VEL
LIN {X 0,Y 80.966,Z 848.847,A -85,B 0,C 180,E1 1170,E2 1170} C_VEL
LIN {X 0,Y 87.976,Z 847.793,A -85,B 0,C 180,E1 1183.807,E2 1183.807} C_VEL
LIN {X 0,Y 99.588,Z 845.033,A -85,B 0,C 180,E1 1194.94,E2 1194.94} C_VEL
LIN {X 0,Y 114.229,Z 840.422,A -85,B 0,C 180,E1 1203.465,E2 1203.465} C_VEL
LIN {X 0,Y 129.592,Z 834.439,A -85,B 0,C 180,E1 1209.543,E2 1209.543} C_VEL
LIN {X 0,Y 147.555,Z 825.922,A -85,B 0,C 180,E1 1214.671,E2 1214.671} C_VEL
LIN {X 0,Y 163.694,Z 816.671,A -85,B 0,C 180,E1 1218.173,E2 1218.173} C_VEL
LIN {X 0,Y 180.982,Z 805.019,A -85,B 0,C 180,E1 1221.165,E2 1221.165} C_VEL
LIN {X 0,Y 196.733,Z 792.471,A -85,B 0,C 180,E1 1223.416,E2 1223.416} C_VEL
LIN {X 0,Y 211.751,Z 778.501,A -85,B 0,C 180,E1 1225.243,E2 1225.243} C_VEL
LIN {X 0,Y 214.564,Z 775.683,A -85,B 0,C 180,E1 1225.532,E2 1225.532} C_VEL
LIN {X 0,Y 222.713,Z 781.532,A -85,B 0,C 180,E1 1219.742,E2 1219.742} C_VEL
LIN {X 0,Y 232.456,Z 788.567,A -85,B 0,C 180,E1 1213.827,E2 1213.827} C_VEL
LIN {X 0,Y 240.138,Z 794.638,A -85,B 0,C 180,E1 1209.261,E2 1209.261} C_VEL
LIN {X 0,Y 243.921,Z 797.459,A -85,B 0,C 180,E1 1206.957,E2 1206.957} C_VEL
LIN {X 0,Y 250.306,Z 802.549,A -85,B 0,C 180,E1 1202.583,E2 1202.583} C_VEL
LIN {X 0,Y 255.293,Z 805.823,A -85,B 0,C 180,E1 1199.173,E2 1199.173} C_VEL
LIN {X 0,Y 259.885,Z 809.878,A -85,B 0,C 180,E1 1195.036,E2 1195.036} C_VEL
LIN {X 0,Y 263.981,Z 812.719,A -85,B 0,C 180,E1 1191.321,E2 1191.321} C_VEL
LIN {X 0,Y 268.443,Z 815.105,A -85,B 0,C 180,E1 1187.112,E2 1187.112} C_VEL
LIN {X 0,Y 270.401,Z 817.339,A -85,B 0,C 180,E1 1183.471,E2 1183.471} C_VEL
LIN {X 0,Y 272.322,Z 819.121,A -85,B 0,C 180,E1 1179.51,E2 1179.51} C_VEL
LIN {X 0,Y 273.679,Z 820.127,A -85,B 0,C 180,E1 1175.661,E2 1175.661} C_VEL
LIN {X 0,Y 274.32,Z 820.576,A -85,B 0,C 180,E1 1172.507,E2 1172.507} C_VEL
LIN {X 0,Y 274.453,Z 820.692,A -85,B 0,C 180,E1 1169.583,E2 1169.583} C_VEL
LIN {X 0,Y 274.178,Z 820.457,A -85,B 0,C 180,E1 1166.446,E2 1166.446} C_VEL
LIN {X 0,Y 273.156,Z 819.792,A -85,B 0,C 180,E1 1162.628,E2 1162.628} C_VEL
LIN {X 0,Y 271.476,Z 818.411,A -85,B 0,C 180,E1 1158.744,E2 1158.744} C_VEL
LIN {X 0,Y 271.021,Z 817.966,A -85,B 0,C 180,E1 1157.747,E2 1157.747} C_VEL
LIN {X 0,Y 269.384,Z 817.694,A -85,B 0,C 180,E1 1156.137,E2 1156.137} C_VEL
LIN {X 0,Y 265.104,Z 818.119,A -85,B 0,C 180,E1 1153.913,E2 1153.913} C_VEL
LIN {X 0,Y 259.771,Z 818.167,A -85,B 0,C 180,E1 1151.171,E2 1151.171} C_VEL
LIN {X 0,Y 258.841,Z 817.772,A -85,B 0,C 180,E1 1150.452,E2 1150.452} C_VEL
LIN {X 0,Y 254.709,Z 815.185,A -85,B 0,C 180,E1 1146.643,E2 1146.643} C_VEL
LIN {X 0,Y 249.764,Z 811.176,A -85,B 0,C 180,E1 1142.186,E2 1142.186} C_VEL
LIN {X 0,Y 247.259,Z 809.168,A -85,B 0,C 180,E1 1140.174,E2 1140.174} C_VEL
LIN {X 0,Y 240.711,Z 804.597,A -85,B 0,C 180,E1 1135.727,E2 1135.727} C_VEL
LIN {X 0,Y 235.421,Z 800.213,A -85,B 0,C 180,E1 1132.159,E2 1132.159} C_VEL
LIN {X 0,Y 226.37,Z 793.394,A -85,B 0,C 180,E1 1126.765,E2 1126.765} C_VEL
LIN {X 0,Y 220.159,Z 789.086,A -85,B 0,C 180,E1 1123.016,E2 1123.016} C_VEL
LIN {X 0,Y 213.535,Z 784.352,A -85,B 0,C 180,E1 1118.5,E2 1118.5} C_VEL
LIN {X 0,Y 211.422,Z 783.274,A -85,B 0,C 180,E1 1117.147,E2 1117.147} C_VEL
LIN {X 0,Y 196.19,Z 796.93,A -85,B 0,C 180,E1 1119.229,E2 1119.229} C_VEL
LIN {X 0,Y 179.907,Z 809.343,A -85,B 0,C 180,E1 1121.867,E2 1121.867} C_VEL
LIN {X 0,Y 163.886,Z 819.788,A -85,B 0,C 180,E1 1125.023,E2 1125.023} C_VEL
LIN {X 0,Y 146.988,Z 829.054,A -85,B 0,C 180,E1 1129.232,E2 1129.232} C_VEL
LIN {X 0,Y 131.69,Z 836.045,A -85,B 0,C 180,E1 1134.225,E2 1134.225} C_VEL
LIN {X 0,Y 115.534,Z 842.153,A -85,B 0,C 180,E1 1141.577,E2 1141.577} C_VEL
LIN {X 0,Y 102.447,Z 846.067,A -85,B 0,C 180,E1 1150.621,E2 1150.621} C_VEL
LIN {X 0,Y 92.409,Z 848.223,A -85,B 0,C 180,E1 1162.54,E2 1162.54} C_VEL
LIN {X 0,Y 89.113,Z 848.606,A -85,B 0,C 180,E1 1170,E2 1170} C_VEL
LIN {X 0,Y 95.96,Z 847.554,A -85,B 0,C 180,E1 1182.639,E2 1182.639} C_VEL
LIN {X 0,Y 107.097,Z 844.788,A -85,B 0,C 180,E1 1193.085,E2 1193.085} C_VEL
LIN {X 0,Y 121.171,Z 840.182,A -85,B 0,C 180,E1 1201.321,E2 1201.321} C_VEL
LIN {X 0,Y 135.613,Z 834.373,A -85,B 0,C 180,E1 1207.197,E2 1207.197} C_VEL
LIN {X 0,Y 152.01,Z 826.45,A -85,B 0,C 180,E1 1212.136,E2 1212.136} C_VEL
LIN {X 0,Y 168.38,Z 816.982,A -85,B 0,C 180,E1 1215.93,E2 1215.93} C_VEL
LIN {X 0,Y 184.402,Z 806.125,A -85,B 0,C 180,E1 1218.908,E2 1218.908} C_VEL
LIN {X 0,Y 199.853,Z 793.84,A -85,B 0,C 180,E1 1221.301,E2 1221.301} C_VEL
LIN {X 0,Y 211.671,Z 783.164,A -85,B 0,C 180,E1 1222.816,E2 1222.816} C_VEL
LIN {X 0,Y 217.014,Z 786.836,A -85,B 0,C 180,E1 1219.076,E2 1219.076} C_VEL
LIN {X 0,Y 225.962,Z 793.051,A -85,B 0,C 180,E1 1213.495,E2 1213.495} C_VEL
LIN {X 0,Y 235.427,Z 800.211,A -85,B 0,C 180,E1 1207.843,E2 1207.843} C_VEL
